LIN {X -165.856,Y 332.396,Z -10.000,A 0.015,B 0.000,C 180.000} C_DIS
LIN {X -166.589,Y 332.890,Z -10.000,A 0.015,B 0.000,C -180.000} C_DIS
LIN {X -177.836,Y 338.486,Z -10.000,A 0.015,B -0.000,C -180.000} C_DIS
LIN {X -178.207,Y 338.644,Z -10.000,A 0.015,B -0.000,C 180.000} C_DIS
LIN {X -178.933,Y 338.902,Z -10.000,A 0.015,B 0.000,C -180.000} C_DIS
LIN {X -179.548,Y 339.058,Z -10.000,A 0.015,B 0.000,C -180.000} C_DIS
LIN {X -180.489,Y 339.204,Z -10.000,A 0.015,B 0.000,C 180.000} C_DIS
LIN {X 4.865,Y 339.209,Z -10.000,A 0.015,B 0.000,C 180.000} C_DIS
LIN {X 5.937,Y 339.152,Z -10.000,A 0.015,B 0.000,C 180.000} C_DIS
LIN {X 6.802,Y 338.955,Z -10.000,A 0.015,B 0.000,C 180.000} C_DIS
LIN {X 7.069,Y 338.840,Z -10.000,A 0.015,B 0.000,C 180.000} C_DIS
LIN {X 7.566,Y 338.456,Z -9.830,A 0.015,B 0.000,C -180.000} C_DIS
LIN {X 7.779,Y 338.046,Z -9.365,A 0.015,B 0.000,C -180.000} C_DIS
LIN {X 7.818,Y 337.880,Z -8.730,A 0.015,B -0.000,C 180.000} C_DIS
$VEL.CP = 1.00000
LIN {X 7.818,Y 337.880,Z 11.000,A 0.015,B -0.000,C 180.000} C_DIS
$VEL.CP = 1.00000
LIN {X 10.265,Y 334.347,Z 11.000,A 0.015,B -0.000,C -180.000} C_DIS
$VEL.CP = 0.10000
LIN {X 10.265,Y 334.347,Z -10.000,A 0.015,B 0.000,C 180.000} C_DIS
LIN {X 10.273,Y 31.575,Z -10.000,A 0.015,B 0.000,C 180.000} C_DIS
LIN {X 8.895,Y 37.171,Z -10.000,A 0.015,B 0.000,C 180.000} C_DIS
LIN {X 8.758,Y 37.599,Z -10.000,A 0.015,B 0.000,C 180.000} C_DIS
LIN {X 8.488,Y 38.288,Z -10.000,A 0.015,B 0.000,C 180.000} C_DIS
LIN {X 8.227,Y 38.812,Z -10.000,A 0.015,B -0.000,C -180.000} C_DIS
LIN {X 2.036,Y 48.951,Z -10.000,A 0.015,B 0.000,C 180.000} C_DIS
LIN {X 1.888,Y 49.173,Z -10.000,A 0.015,B -0.000,C 180.000} C_DIS
LIN {X 1.052,Y 50.326,Z -10.000,A 0.015,B 0.000,C -180.000} C_DIS
LIN {X 0.431,Y 50.979,Z -10.000,A 0.015,B 0.000,C 180.000} C_DIS
LIN {X -7.440,Y 57.297,Z -10.000,A 0.015,B 0.000,C -180.000} C_DIS
LIN {X -7.815,Y 57.559,Z -10.000,A 0.015,B 0.000,C 180.000} C_DIS
LIN {X -8.485,Y 57.962,Z -10.000,A 0.015,B 0.000,C -180.000} C_DIS
LIN {X -9.252,Y 58.301,Z -10.000,A 0.015,B 0.000,C 180.000} C_DIS
LIN {X -19.103,Y 61.267,Z -10.000,A 0.015,B 0.000,C -180.000} C_DIS
LIN {X -19.948,Y 61.408,Z -10.000,A 0.015,B -0.000,C -180.000} C_DIS
LIN {X -21.762,Y 61.478,Z -10.000,A 0.015,B 0.000,C -180.000} C_DIS
LIN {X -22.200,Y 61.466,Z -10.000,A 0.015,B -0.000,C -180.000} C_DIS
LIN {X -29.456,Y 60.802,Z -10.000,A 0.015,B -0.000,C -180.000} C_DIS
LIN {X -29.688,Y 60.773,Z -10.000,A 0.015,B 0.000,C 180.000} C_DIS
LIN {X -31.502,Y 60.480,Z -10.000,A 0.015,B 0.000,C 180.000} C_DIS
LIN {X -32.206,Y 60.286,Z -10.000,A 0.015,B 0.000,C 180.000} C_DIS
LIN {X -34.020,Y 59.568,Z -10.000,A 0.015,B 0.000,C 180.000} C_DIS
LIN {X -34.313,Y 59.436,Z -10.000,A 0.015,B 0.000,C 180.000} C_DIS
LIN {X -41.056,Y 55.994,Z -10.000,A 0.015,B 0.000,C -180.000} C_DIS
LIN {X -41.306,Y 55.853,Z -10.000,A 0.015,B 0.000,C -180.000} C_DIS
LIN {X -42.245,Y 55.268,Z -10.000,A 0.015,B 0.000,C 180.000} C_DIS
LIN {X -42.603,Y 55.011,Z -10.000,A 0.015,B -0.000,C 180.000} C_DIS
LIN {X -43.629,Y 54.169,Z -10.000,A 0.015,B 0.000,C 180.000} C_DIS
LIN {X -44.021,Y 53.790,Z -10.000,A 0.015,B -0.000,C 180.000} C_DIS
LIN {X -46.923,Y 50.493,Z -10.000,A 0.015,B 0.000,C -180.000} C_DIS
LIN {X -46.984,Y 50.423,Z -10.000,A 0.015,B 0.000,C -180.000} C_DIS
LIN {X -50.315,Y 46.422,Z -10.000,A 0.015,B 0.000,C -180.000} C_DIS
LIN {X -50.645,Y 45.950,Z -10.000,A 0.015,B 0.000,C -180.000} C_DIS
LIN {X -68.582,Y 14.913,Z -10.000,A 0.015,B 0.000,C -180.000} C_DIS
LIN {X -68.710,Y 14.669,Z -10.000,A 0.015,B -0.000,C 180.000} C_DIS
LIN {X -69.398,Y 13.218,Z -10.000,A 0.015,B 0.000,C 180.000} C_DIS
LIN {X -69.532,Y 12.892,Z -10.000,A 0.015,B 0.000,C 180.000} C_DIS
LIN {X -72.086,Y 5.638,Z -10.000,A 0.015,B 0.000,C 180.000} C_DIS
LIN {X -72.157,Y 5.411,Z -10.000,A 0.015,B 0.000,C -180.000} C_DIS
LIN {X -72.555,Y 3.960,Z -10.000,A 0.015,B 0.000,C -180.000} C_DIS
LIN {X -72.656,Y 3.432,Z -10.000,A 0.015,B 0.000,C 180.000} C_DIS
LIN {X -72.815,Y 1.981,Z -10.000,A 0.015,B 0.000,C -180.000} C_DIS
LIN {X -72.832,Y 1.451,Z -10.000,A 0.015,B 0.000,C -180.000} C_DIS
LIN {X -72.484,Y -5.804,Z -10.000,A 0.015,B -0.000,C 180.000} C_DIS
LIN {X -72.471,Y -5.978,Z -10.000,A 0.015,B 0.000,C 180.000} C_DIS
LIN {X -72.255,Y -8.154,Z -10.000,A 0.015,B 0.000,C -180.000} C_DIS
LIN {X -72.121,Y -8.815,Z -10.000,A 0.015,B 0.000,C -180.000} C_DIS
LIN {X -71.696,Y -10.196,Z -10.000,A 0.015,B 0.000,C 180.000} C_DIS
LIN {X -71.562,Y -10.556,Z -10.000,A 0.015,B 0.000,C -180.000} C_DIS
LIN {X -70.702,Y -12.522,Z -10.000,A 0.015,B 0.000,C -180.000} C_DIS
LIN {X -70.675,Y -12.581,Z -10.000,A 0.015,B -0.000,C 180.000} C_DIS
LIN {X -68.540,Y -17.215,Z -10.000,A 0.015,B 0.000,C 180.000} C_DIS
LIN {X -68.479,Y -17.341,Z -10.000,A 0.015,B 0.000,C -180.000} C_DIS
LIN {X -67.736,Y -18.792,Z -10.000,A 0.015,B 0.000,C 180.000} C_DIS
LIN {X -67.504,Y -19.179,Z -10.000,A 0.015,B 0.000,C -180.000} C_DIS
LIN {X -66.730,Y -20.294,Z -10.000,A 0.015,B 0.000,C -180.000} C_DIS
LIN {X -66.274,Y -20.824,Z -10.000,A 0.015,B -0.000,C 180.000} C_DIS
LIN {X -59.767,Y -26.968,Z -10.000,A 0.015,B 0.000,C 180.000} C_DIS
LIN {X -59.610,Y -27.107,Z -10.000,A 0.015,B 0.000,C 180.000} C_DIS
LIN {X -58.521,Y -28.014,Z -10.000,A 0.015,B 0.000,C 180.000} C_DIS
CIRC {X -58.086,Y -28.321,Z -10.000,A 0.015,B 0.000,C 180.000},{X -57.609,Y -28.557,Z -10.000,A 0.015,B 0.000,C 180.000} C_DIS
LIN {X -50.808,Y -31.266,Z -10.000,A 0.015,B 0.000,C 180.000} C_DIS
LIN {X -342.732,Y -31.266,Z -10.000,A 0.015,B 0.000,C -180.000} C_DIS
LIN {X -336.289,Y -28.753,Z -10.000,A 0.015,B 0.000,C 180.000} C_DIS
LIN {X -335.780,Y -28.504,Z -10.000,A 0.015,B -0.000,C 180.000} C_DIS
LIN {X -335.055,Y -28.070,Z -10.000,A 0.015,B 0.000,C -180.000} C_DIS
LIN {X -334.490,Y -27.645,Z -10.000,A 0.015,B -0.000,C -180.000} C_DIS
LIN {X -332.313,Y -25.623,Z -10.000,A 0.015,B 0.000,C 180.000} C_DIS
LIN {X -332.274,Y -25.586,Z -10.000,A 0.015,B -0.000,C -180.000} C_DIS
LIN {X -326.917,Y -20.448,Z -10.000,A 0.015,B 0.000,C 180.000} C_DIS
LIN {X -326.374,Y -19.773,Z -10.000,A 0.015,B -0.000,C 180.000} C_DIS
LIN {X -325.688,Y -18.654,Z -10.000,A 0.015,B -0.000,C 180.000} C_DIS
LIN {X -325.506,Y -18.313,Z -10.000,A 0.015,B 0.000,C 180.000} C_DIS
LIN {X -322.238,Y -11.280,Z -10.000,A 0.015,B 0.000,C 180.000} C_DIS
LIN {X -322.125,Y -11.006,Z -10.000,A 0.015,B 0.000,C -180.000} C_DIS
LIN {X -321.519,Y -9.333,Z -10.000,A 0.015,B 0.000,C -180.000} C_DIS
LIN {X -321.339,Y -8.569,Z -10.000,A 0.015,B -0.000,C -180.000} C_DIS
LIN {X -321.046,Y -6.030,Z -10.000,A 0.015,B 0.000,C -180.000} C_DIS
LIN {X -321.028,Y -5.804,Z -10.000,A 0.015,B -0.000,C -180.000} C_DIS
LIN {X -320.680,Y 1.451,Z -10.000,A 0.015,B 0.000,C 180.000} C_DIS
LIN {X -320.686,Y 1.861,Z -10.000,A 0.015,B 0.000,C -180.000} C_DIS
LIN {X -320.739,Y 2.586,Z -10.000,A 0.015,B -0.000,C -180.000} C_DIS
LIN {X -320.784,Y 2.941,Z -10.000,A 0.015,B -0.000,C -180.000} C_DIS
LIN {X -321.047,Y 4.392,Z -10.000,A 0.015,B -0.000,C 180.000} C_DIS
LIN {X -321.174,Y 4.882,Z -10.000,A 0.015,B 0.000,C -180.000} C_DIS
LIN {X -321.917,Y 7.058,Z -10.000,A 0.015,B 0.000,C 180.000} C_DIS
LIN {X -321.936,Y 7.114,Z -10.000,A 0.015,B -0.000,C 180.000} C_DIS
LIN {X -324.293,Y 13.643,Z -10.000,A 0.015,B 0.000,C 180.000} C_DIS
LIN {X -324.544,Y 14.184,Z -10.000,A 0.015,B 0.000,C -180.000} C_DIS
LIN {X -342.520,Y 45.380,Z -10.000,A 0.015,B -0.000,C -180.000} C_DIS
LIN {X -342.658,Y 45.599,Z -10.000,A 0.015,B 0.000,C 180.000} C_DIS
LIN {X -343.432,Y 46.732,Z -10.000,A 0.015,B -0.000,C 180.000} C_DIS
LIN {X -343.654,Y 47.022,Z -10.000,A 0.015,B 0.000,C -180.000} C_DIS
LIN {X -348.970,Y 53.238,Z -10.000,A 0.015,B 0.000,C 180.000} C_DIS
LIN {X -349.184,Y 53.466,Z -10.000,A 0.015,B 0.000,C 180.000} C_DIS
LIN {X -350.186,Y 54.439,Z -10.000,A 0.015,B 0.000,C 180.000} C_DIS
LIN {X -350.569,Y 54.760,Z -10.000,A 0.015,B 0.000,C -180.000} C_DIS
LIN {X -351.551,Y 55.465,Z -10.000,A 0.015,B 0.000,C 180.000} C_DIS
LIN {X -351.978,Y 55.726,Z -10.000,A 0.015,B 0.000,C -180.000} C_DIS
LIN {X -359.191,Y 59.432,Z -10.000,A 0.015,B 0.000,C -180.000} C_DIS
LIN {X -359.413,Y 59.536,Z -10.000,A 0.015,B 0.000,C -180.000} C_DIS
LIN {X -360.864,Y 60.153,Z -10.000,A 0.015,B -0.000,C 180.000} C_DIS
LIN {X -361.495,Y 60.351,Z -10.000,A 0.015,B 0.000,C -180.000} C_DIS
LIN {X -362.947,Y 60.654,Z -10.000,A 0.015,B 0.000,C 180.000} C_DIS
LIN {X -363.320,Y 60.711,Z -10.000,A 0.015,B 0.000,C 180.000} C_DIS
LIN {X -371.302,Y 61.465,Z -10.000,A 0.015,B 0.000,C -180.000} C_DIS
LIN {X -371.750,Y 61.478,Z -10.000,A 0.015,B 0.000,C -180.000} C_DIS
LIN {X -373.564,Y 61.408,Z -10.000,A 0.015,B -0.000,C 180.000} C_DIS
LIN {X -374.398,Y 61.270,Z -10.000,A 0.015,B -0.000,C -180.000} C_DIS
LIN {X -383.578,Y 58.541,Z -10.000,A 0.015,B 0.000,C -180.000} C_DIS
LIN {X -383.897,Y 58.428,Z -10.000,A 0.015,B 0.000,C 180.000} C_DIS
LIN {X -384.902,Y 58.016,Z -10.000,A 0.015,B 0.000,C 180.000} C_DIS
LIN {X -385.717,Y 57.540,Z -10.000,A 0.015,B -0.000,C 180.000} C_DIS
LIN {X -393.232,Y 51.598,Z -10.000,A 0.015,B 0.000,C -180.000} C_DIS
LIN {X -393.470,Y 51.391,Z -10.000,A 0.015,B -0.000,C 180.000} C_DIS
LIN {X -394.404,Y 50.499,Z -10.000,A 0.015,B 0.000,C -180.000} C_DIS
LIN {X -394.942,Y 49.837,Z -10.000,A 0.015,B -0.000,C 180.000} C_DIS
LIN {X -401.253,Y 39.671,Z -10.000,A 0.015,B 0.000,C 180.000} C_DIS
LIN {X -401.377,Y 39.454,Z -10.000,A 0.015,B 0.000,C 180.000} C_DIS
LIN {X -401.994,Y 38.272,Z -10.000,A 0.015,B 0.000,C -180.000} C_DIS
LIN {X -402.274,Y 37.542,Z -10.000,A 0.015,B -0.000,C 180.000} C_DIS
LIN {X -403.779,Y 31.645,Z -10.000,A 0.015,B 0.000,C 180.000} C_DIS
LIN {X -403.787,Y 333.800,Z -10.000,A 0.015,B 0.000,C 180.000} C_DIS
LIN {X -403.730,Y 334.871,Z -10.000,A 0.015,B -0.000,C -180.000} C_DIS
LIN {X -403.533,Y 335.736,Z -10.000,A 0.015,B 0.000,C -180.000} C_DIS
LIN {X -403.418,Y 336.003,Z -10.000,A 0.015,B -0.000,C -180.000} C_DIS
LIN {X -403.034,Y 336.500,Z -9.830,A 0.015,B 0.000,C -180.000} C_DIS
LIN {X -402.624,Y 336.714,Z -9.365,A 0.015,B -0.000,C -180.000} C_DIS
LIN {X -402.458,Y 336.753,Z -8.730,A 0.015,B 0.000,C -180.000} C_DIS
$VEL.CP = 1.00000
LIN {X -402.458,Y 336.753,Z 11.000,A 0.015,B 0.000,C 180.000} C_DIS
$VEL.CP = 1.00000
LIN {X -182.199,Y 109.361,Z 11.000,A 0.015,B 0.000,C 180.000} C_DIS
$VEL.CP = 1.00000
LIN {X -182.199,Y 109.361,Z 1.769,A 0.015,B -0.000,C 180.000} C_DIS
$VEL.CP = 0.10000
LIN {X -182.037,Y 109.343,Z 1.147,A 0.015,B 0.000,C 180.000} C_DIS
LIN {X -181.592,Y 109.314,Z 0.684,A 0.015,B -0.000,C -180.000} C_DIS
LIN {X -180.976,Y 109.330,Z 0.500,A 0.015,B 0.000,C -180.000} C_DIS
LIN {X -175.739,Y 113.354,Z 0.256,A 0.015,B 0.000,C -180.000} C_DIS
LIN {X -177.328,Y 119.764,Z 0.012,A 0.015,B 0.000,C 180.000} C_DIS
LIN {X -183.837,Y 120.878,Z -0.232,A 0.015,B 0.000,C -180.000} C_DIS
LIN {X -187.466,Y 115.360,Z -0.476,A 0.015,B -0.000,C -180.000} C_DIS
LIN {X -183.865,Y 109.824,Z -0.720,A 0.015,B 0.000,C -180.000} C_DIS
LIN {X -177.349,Y 110.905,Z -0.964,A 0.015,B 0.000,C -180.000} C_DIS
LIN {X -175.729,Y 117.308,Z -1.208,A 0.015,B 0.000,C -180.000} C_DIS
LIN {X -180.946,Y 121.358,Z -1.452,A 0.015,B 0.000,C -180.000} C_DIS
LIN {X -186.747,Y 118.201,Z -1.696,A 0.015,B 0.000,C -180.000} C_DIS
LIN {X -186.180,Y 111.621,Z -1.940,A 0.015,B 0.000,C -180.000} C_DIS
LIN {X -179.924,Y 109.504,Z -2.185,A 0.015,B 0.000,C 180.000} C_DIS
LIN {X -175.478,Y 114.388,Z -2.429,A 0.015,B -0.000,C -180.000} C_DIS
LIN {X -178.170,Y 120.418,Z -2.673,A 0.015,B 0.000,C 180.000} C_DIS
LIN {X -184.774,Y 120.368,Z -2.917,A 0.015,B 0.000,C 180.000} C_DIS
LIN {X -187.374,Y 114.297,Z -3.161,A 0.015,B -0.000,C 180.000} C_DIS
LIN {X -182.854,Y 109.482,Z -3.405,A 0.015,B 0.000,C -180.000} C_DIS
LIN {X -176.631,Y 111.694,Z -3.649,A 0.015,B 0.000,C -180.000} C_DIS
LIN {X -176.164,Y 118.282,Z -3.893,A 0.015,B 0.000,C 180.000} C_DIS
LIN {X -182.013,Y 121.350,Z -4.137,A 0.015,B 0.000,C 180.000} C_DIS
LIN {X -187.167,Y 117.220,Z -4.381,A 0.015,B 0.000,C -180.000} C_DIS
LIN {X -185.449,Y 110.843,Z -4.625,A 0.015,B 0.000,C 180.000} C_DIS
LIN {X -178.919,Y 109.862,Z -4.869,A 0.015,B -0.000,C -180.000} C_DIS
LIN {X -175.402,Y 115.452,Z -5.113,A 0.015,B 0.000,C 180.000} C_DIS
LIN {X -179.115,Y 120.914,Z -5.357,A 0.015,B 0.000,C -180.000} C_DIS
LIN {X -185.607,Y 119.701,Z -5.601,A 0.015,B 0.000,C 180.000} C_DIS
LIN {X -187.097,Y 113.267,Z -5.845,A 0.015,B 0.000,C -180.000} C_DIS
LIN {X -181.799,Y 109.324,Z -6.089,A 0.015,B 0.000,C -180.000} C_DIS
LIN {X -176.063,Y 112.597,Z -6.333,A 0.015,B 0.000,C -180.000} C_DIS
LIN {X -176.764,Y 119.164,Z -6.577,A 0.015,B 0.000,C -180.000} C_DIS
LIN {X -183.061,Y 121.154,Z -6.821,A 0.015,B 0.000,C 180.000} C_DIS
LIN {X -187.408,Y 116.181,Z -7.065,A 0.015,B 0.000,C 180.000} C_DIS
LIN {X -184.594,Y 110.206,Z -7.310,A 0.015,B 0.000,C -180.000} C_DIS
LIN {X -177.992,Y 110.390,Z -7.554,A 0.015,B 0.000,C -180.000} C_DIS
LIN {X -175.515,Y 116.513,Z -7.798,A 0.015,B -0.000,C 180.000} C_DIS
LIN {X -180.132,Y 121.235,Z -8.042,A 0.015,B 0.000,C -180.000} C_DIS
LIN {X -186.309,Y 118.898,Z -8.286,A 0.015,B 0.000,C 180.000} C_DIS
LIN {X -186.643,Y 112.302,Z -8.530,A 0.015,B -0.000,C 180.000} C_DIS
LIN {X -180.733,Y 109.353,Z -8.774,A 0.015,B 0.000,C 180.000} C_DIS
LIN {X -175.663,Y 113.586,Z -9.018,A 0.015,B -0.000,C -180.000} C_DIS
LIN {X -177.510,Y 119.927,Z -9.262,A 0.015,B 0.000,C 180.000} C_DIS
LIN {X -184.059,Y 120.776,Z -9.506,A 0.015,B 0.000,C -180.000} C_DIS
LIN {X -187.462,Y 115.116,Z -9.750,A 0.015,B 0.000,C -180.000} C_DIS
LIN {X -183.639,Y 109.730,Z -9.994,A 0.015,B 0.000,C 180.000} C_DIS
LIN {X -177.173,Y 111.074,Z -10.238,A 0.015,B 0.000,C 180.000} C_DIS
LIN {X -175.813,Y 117.537,Z -10.482,A 0.015,B 0.000,C 180.000} C_DIS
LIN {X -181.190,Y 121.373,Z -10.726,A 0.015,B 0.000,C -180.000} C_DIS
LIN {X -186.858,Y 117.984,Z -10.970,A 0.015,B 0.000,C 180.000} C_DIS
LIN {X -186.025,Y 111.432,Z -11.214,A 0.015,B -0.000,C -180.000} C_DIS
LIN {X -179.689,Y 109.570,Z -11.458,A 0.015,B 0.000,C -180.000} C_DIS
LIN {X -175.444,Y 114.630,Z -11.702,A 0.015,B 0.000,C 180.000} C_DIS
LIN {X -178.378,Y 120.546,Z -11.946,A 0.015,B 0.000,C -180.000} C_DIS
LIN {X -184.975,Y 120.229,Z -12.190,A 0.015,B 0.000,C 180.000} C_DIS
LIN {X -187.327,Y 114.058,Z -12.435,A 0.015,B -0.000,C -180.000} C_DIS
LIN {X -182.616,Y 109.429,Z -12.679,A 0.015,B -0.000,C -180.000} C_DIS
LIN {X -176.488,Y 111.891,Z -12.923,A 0.015,B -0.000,C -180.000} C_DIS
LIN {X -176.287,Y 118.492,Z -13.167,A 0.015,B 0.000,C 180.000} C_DIS
LIN {X -182.255,Y 121.321,Z -13.411,A 0.015,B 0.000,C -180.000} C_DIS
LIN {X -187.238,Y 116.987,Z -13.655,A 0.015,B 0.000,C 180.000} C_DIS
LIN {X -185.264,Y 110.685,Z -13.899,A 0.015,B -0.000,C -180.000} C_DIS
LIN {X -178.699,Y 109.968,Z -14.143,A 0.015,B 0.000,C -180.000} C_DIS
LIN {X -175.411,Y 115.696,Z -14.387,A 0.015,B -0.000,C 180.000} C_DIS
LIN {X -179.342,Y 121.003,Z -14.631,A 0.015,B -0.000,C 180.000} C_DIS
LIN {X -185.780,Y 119.529,Z -14.875,A 0.015,B 0.000,C -180.000} C_DIS
LIN {X -187.008,Y 113.040,Z -15.119,A 0.015,B -0.000,C 180.000} C_DIS
LIN {X -181.556,Y 109.314,Z -15.363,A 0.015,B 0.000,C 180.000} C_DIS
LIN {X -175.957,Y 112.816,Z -15.607,A 0.015,B 0.000,C -180.000} C_DIS
LIN {X -176.922,Y 119.350,Z -15.851,A 0.015,B -0.000,C -180.000} C_DIS
LIN {X -183.295,Y 121.083,Z -16.095,A 0.015,B 0.000,C 180.000} C_DIS
LIN {X -187.437,Y 115.939,Z -16.339,A 0.015,B 0.000,C 180.000} C_DIS
LIN {X -184.384,Y 110.083,Z -16.583,A 0.015,B -0.000,C 180.000} C_DIS
LIN {X -177.795,Y 110.534,Z -16.827,A 0.015,B 0.000,C 180.000} C_DIS
LIN {X -175.567,Y 116.751,Z -17.071,A 0.015,B 0.000,C -180.000} C_DIS
LIN {X -180.371,Y 121.283,Z -17.315,A 0.015,B -0.000,C 180.000} C_DIS
LIN {X -186.448,Y 118.698,Z -17.560,A 0.015,B 0.000,C -180.000} C_DIS
LIN {X -186.515,Y 112.094,Z -17.804,A 0.015,B 0.000,C -180.000} C_DIS
LIN {X -180.491,Y 109.386,Z -18.048,A 0.015,B -0.000,C 180.000} C_DIS
LIN {X -175.597,Y 113.821,Z -18.292,A 0.015,B 0.000,C -180.000} C_DIS
LIN {X -177.698,Y 120.082,Z -18.536,A 0.015,B 0.000,C 180.000} C_DIS
LIN {X -184.277,Y 120.666,Z -18.780,A 0.015,B -0.000,C 180.000} C_DIS
LIN {X -187.448,Y 114.872,Z -19.024,A 0.015,B 0.000,C 180.000} C_DIS
LIN {X -183.411,Y 109.646,Z -19.268,A 0.015,B -0.000,C -180.000} C_DIS
LIN {X -177.004,Y 111.250,Z -19.512,A 0.015,B -0.000,C 180.000} C_DIS
LIN {X -175.907,Y 117.762,Z -19.756,A 0.015,B 0.000,C 180.000} C_DIS
LIN {X -181.434,Y 121.377,Z -20.000,A 0.015,B 0.000,C -180.000} C_DIS
LIN {X -213.976,Y 121.377,Z -20.000,A 0.015,B 0.000,C 180.000} C_DIS
CIRC {X -215.901,Y 120.266,Z -20.000,A 0.015,B 0.000,C 180.000},{X -215.902,Y 118.044,Z -20.000,A 0.015,B 0.000,C -180.000} C_DIS
LIN {X -214.807,Y 116.142,Z -20.000,A 0.015,B 0.000,C 180.000} C_DIS
CIRC {X -213.767,Y 115.102,Z -20.000,A 0.015,B 0.000,C 180.000},{X -212.347,Y 114.721,Z -20.000,A 0.015,B 0.000,C -180.000} C_DIS
LIN {X -181.151,Y 114.721,Z -20.000,A 0.015,B 0.000,C 180.000} C_DIS
CIRC {X -179.732,Y 115.101,Z -20.000,A 0.015,B 0.000,C 180.000},{X -178.693,Y 116.139,Z -20.000,A 0.015,B 0.000,C 180.000} C_DIS
LIN {X -177.595,Y 118.039,Z -20.000,A 0.015,B -0.000,C 180.000} C_DIS
CIRC {X -177.595,Y 120.265,Z -20.000,A 0.015,B 0.000,C 180.000},{X -179.522,Y 121.377,Z -20.000,A 0.015,B -0.000,C 180.000} C_DIS
LIN {X -181.434,Y 121.377,Z -20.000,A 0.015,B 0.000,C -180.000} C_DIS
CIRC {X -184.808,Y 122.399,Z -20.000,A 0.015,B 0.000,C 180.000},{X -187.049,Y 125.121,Z -20.000,A 0.015,B 0.000,C 180.000} C_DIS
CIRC {X -189.290,Y 127.843,Z -20.000,A 0.015,B 0.000,C 180.000},{X -192.665,Y 128.864,Z -20.000,A 0.015,B 0.000,C 180.000} C_DIS
LIN {X -214.895,Y 128.864,Z -20.000,A 0.015,B -0.000,C 180.000} C_DIS
CIRC {X -218.571,Y 128.969,Z -20.000,A 0.015,B 0.000,C -180.000},{X -222.234,Y 129.283,Z -20.000,A 0.015,B 0.000,C -180.000} C_DIS
CIRC {X -225.886,Y 129.692,Z -20.000,A 0.015,B 0.000,C 180.000},{X -229.541,Y 130.082,Z -20.000,A 0.015,B 0.000,C 180.000} C_DIS
CIRC {X -231.339,Y 129.164,Z -20.000,A 0.015,B 0.000,C -180.000},{X -231.232,Y 127.147,Z -20.000,A 0.015,B 0.000,C -180.000} C_DIS
CIRC {X -228.499,Y 123.234,Z -20.000,A 0.015,B 0.000,C 180.000},{X -225.916,Y 119.220,Z -20.000,A 0.015,B 0.000,C 180.000} C_DIS
CIRC {X -223.440,Y 115.140,Z -20.000,A 0.015,B 0.000,C 180.000},{X -221.026,Y 111.023,Z -20.000,A 0.015,B -0.000,C 180.000} C_DIS
CIRC {X -217.921,Y 107.915,Z -20.000,A 0.015,B 0.000,C 180.000},{X -213.677,Y 106.777,Z -20.000,A 0.015,B -0.000,C 180.000} C_DIS
LIN {X -179.835,Y 106.777,Z -20.000,A 0.015,B 0.000,C -180.000} C_DIS
CIRC {X -175.585,Y 107.915,Z -20.000,A 0.015,B -0.000,C -180.000},{X -172.474,Y 111.024,Z -20.000,A 0.015,B 0.000,C 180.000} C_DIS
CIRC {X -170.062,Y 115.134,Z -20.000,A 0.015,B 0.000,C -180.000},{X -167.597,Y 119.212,Z -20.000,A 0.015,B 0.000,C -180.000} C_DIS
CIRC {X -165.028,Y 123.227,Z -20.000,A 0.015,B -0.000,C 180.000},{X -162.308,Y 127.141,Z -20.000,A 0.015,B 0.000,C 180.000} C_DIS
CIRC {X -162.205,Y 129.160,Z -20.000,A 0.015,B 0.000,C 180.000},{X -164.006,Y 130.079,Z -20.000,A 0.015,B -0.000,C 180.000} C_DIS
CIRC {X -167.652,Y 129.690,Z -20.000,A 0.015,B -0.000,C 180.000},{X -171.295,Y 129.283,Z -20.000,A 0.015,B 0.000,C 180.000} C_DIS
CIRC {X -174.950,Y 128.969,Z -20.000,A 0.015,B -0.000,C 180.000},{X -178.617,Y 128.865,Z -20.000,A 0.015,B 0.000,C -180.000} C_DIS
LIN {X -192.665,Y 128.864,Z -20.000,A 0.015,B 0.000,C -180.000} C_DIS
CIRC {X -195.950,Y 129.859,Z -20.000,A 0.015,B 0.000,C -180.000},{X -198.132,Y 132.509,Z -20.000,A 0.015,B 0.000,C 180.000} C_DIS
CIRC {X -200.314,Y 135.159,Z -20.000,A 0.015,B 0.000,C 180.000},{X -203.599,Y 136.154,Z -20.000,A 0.015,B 0.000,C 180.000} C_DIS
LIN {X -214.895,Y 136.154,Z -20.000,A 0.015,B 0.000,C -180.000} C_DIS
CIRC {X -223.130,Y 136.478,Z -20.000,A 0.015,B 0.000,C 180.000},{X -231.314,Y 137.447,Z -20.000,A 0.015,B -0.000,C -180.000} C_DIS
CIRC {X -239.436,Y 138.810,Z -20.000,A 0.015,B 0.000,C -180.000},{X -247.532,Y 140.318,Z -20.000,A 0.015,B -0.000,C 180.000} C_DIS
CIRC {X -249.264,Y 139.531,Z -20.000,A 0.015,B 0.000,C 180.000},{X -249.086,Y 137.637,Z -20.000,A 0.015,B -0.000,C 180.000} C_DIS
CIRC {X -243.729,Y 131.288,Z -20.000,A 0.015,B -0.000,C 180.000},{X -238.530,Y 124.808,Z -20.000,A 0.015,B 0.000,C 180.000} C_DIS
CIRC {X -233.643,Y 118.085,Z -20.000,A 0.015,B 0.000,C -180.000},{X -229.242,Y 111.034,Z -20.000,A 0.015,B 0.000,C 180.000} C_DIS
CIRC {X -228.225,Y 109.203,Z -20.000,A 0.015,B 0.000,C -180.000},{X -227.265,Y 107.341,Z -20.000,A 0.015,B 0.000,C -180.000} C_DIS
CIRC {X -226.305,Y 105.479,Z -20.000,A 0.015,B 0.000,C 180.000},{X -225.288,Y 103.648,Z -20.000,A 0.015,B 0.000,C 180.000} C_DIS
CIRC {X -222.183,Y 100.539,Z -20.000,A 0.015,B 0.000,C -180.000},{X -217.939,Y 99.401,Z -20.000,A 0.015,B -0.000,C -180.000} C_DIS
LIN {X -175.579,Y 99.401,Z -20.000,A 0.015,B 0.000,C 180.000} C_DIS
CIRC {X -171.329,Y 100.540,Z -20.000,A 0.015,B -0.000,C 180.000},{X -168.218,Y 103.649,Z -20.000,A 0.015,B 0.000,C -180.000} C_DIS
CIRC {X -167.137,Y 105.588,Z -20.000,A 0.015,B 0.000,C -180.000},{X -166.118,Y 107.559,Z -20.000,A 0.015,B 0.000,C -180.000} C_DIS
CIRC {X -165.099,Y 109.531,Z -20.000,A 0.015,B 0.000,C 180.000},{X -164.019,Y 111.469,Z -20.000,A 0.015,B -0.000,C -180.000} C_DIS
CIRC {X -159.670,Y 118.415,Z -20.000,A 0.015,B 0.000,C 180.000},{X -154.841,Y 125.037,Z -20.000,A 0.015,B 0.000,C 180.000} C_DIS
CIRC {X -149.698,Y 131.412,Z -20.000,A 0.015,B 0.000,C 180.000},{X -144.387,Y 137.648,Z -20.000,A 0.015,B 0.000,C 180.000} C_DIS
CIRC {X -144.201,Y 139.539,Z -20.000,A 0.015,B 0.000,C 180.000},{X -145.931,Y 140.327,Z -20.000,A 0.015,B 0.000,C -180.000} C_DIS
CIRC {X -154.039,Y 138.817,Z -20.000,A 0.015,B 0.000,C 180.000},{X -162.173,Y 137.451,Z -20.000,A 0.015,B 0.000,C 180.000} C_DIS
CIRC {X -170.369,Y 136.479,Z -20.000,A 0.015,B -0.000,C -180.000},{X -178.617,Y 136.154,Z -20.000,A 0.015,B -0.000,C -180.000} C_DIS
LIN {X -203.599,Y 136.154,Z -20.000,A 0.015,B 0.000,C 180.000} C_DIS
CIRC {X -206.696,Y 137.092,Z -20.000,A 0.015,B 0.000,C 180.000},{X -208.752,Y 139.589,Z -20.000,A 0.015,B -0.000,C 180.000} C_DIS
CIRC {X -210.808,Y 142.086,Z -20.000,A 0.015,B 0.000,C -180.000},{X -213.904,Y 143.024,Z -20.000,A 0.015,B -0.000,C 180.000} C_DIS
LIN {X -214.895,Y 143.024,Z -20.000,A 0.015,B -0.000,C -180.000} C_DIS
CIRC {X -230.200,Y 143.852,Z -20.000,A 0.015,B -0.000,C 180.000},{X -245.325,Y 146.329,Z -20.000,A 0.015,B 0.000,C 180.000} C_DIS
CIRC {X -260.127,Y 150.280,Z -20.000,A 0.015,B 0.000,C -180.000},{X -274.518,Y 155.531,Z -20.000,A 0.015,B 0.000,C -180.000} C_DIS
CIRC {X -276.076,Y 155.002,Z -20.000,A 0.015,B 0.000,C 180.000},{X -275.748,Y 153.390,Z -20.000,A 0.015,B 0.000,C 180.000} C_DIS
CIRC {X -266.780,Y 146.054,Z -20.000,A 0.015,B 0.000,C 180.000},{X -258.385,Y 138.068,Z -20.000,A 0.015,B -0.000,C -180.000} C_DIS
CIRC {X -250.572,Y 129.516,Z -20.000,A 0.015,B 0.000,C -180.000},{X -243.334,Y 120.471,Z -20.000,A 0.015,B -0.000,C 180.000} C_DIS
CIRC {X -241.113,Y 117.375,Z -20.000,A 0.015,B 0.000,C 180.000},{X -239.019,Y 114.192,Z -20.000,A 0.015,B 0.000,C 180.000} C_DIS
CIRC {X -237.021,Y 110.948,Z -20.000,A 0.015,B 0.000,C 180.000},{X -235.087,Y 107.666,Z -20.000,A 0.015,B 0.000,C -180.000} C_DIS
CIRC {X -233.587,Y 104.967,Z -20.000,A 0.015,B 0.000,C -180.000},{X -232.172,Y 102.222,Z -20.000,A 0.015,B 0.000,C -180.000} C_DIS
CIRC {X -230.758,Y 99.478,Z -20.000,A 0.015,B 0.000,C 180.000},{X -229.258,Y 96.779,Z -20.000,A 0.015,B 0.000,C -180.000} C_DIS
CIRC {X -226.153,Y 93.670,Z -20.000,A 0.015,B 0.000,C 180.000},{X -221.909,Y 92.532,Z -20.000,A 0.015,B 0.000,C 180.000} C_DIS
LIN {X -171.614,Y 92.532,Z -20.000,A 0.015,B -0.000,C 180.000} C_DIS
CIRC {X -167.365,Y 93.670,Z -20.000,A 0.015,B -0.000,C 180.000},{X -164.253,Y 96.779,Z -20.000,A 0.015,B 0.000,C 180.000} C_DIS
CIRC {X -162.690,Y 99.584,Z -20.000,A 0.015,B -0.000,C -180.000},{X -161.216,Y 102.437,Z -20.000,A 0.015,B 0.000,C -180.000} C_DIS
CIRC {X -159.741,Y 105.289,Z -20.000,A 0.015,B 0.000,C -180.000},{X -158.178,Y 108.094,Z -20.000,A 0.015,B 0.000,C 180.000} C_DIS
CIRC {X -149.836,Y 120.906,Z -20.000,A 0.015,B 0.000,C -180.000},{X -140.182,Y 132.761,Z -20.000,A 0.015,B 0.000,C 180.000} C_DIS
CIRC {X -129.413,Y 143.604,Z -20.000,A 0.015,B -0.000,C -180.000},{X -117.706,Y 153.428,Z -20.000,A 0.015,B 0.000,C 180.000} C_DIS
CIRC {X -117.387,Y 155.041,Z -20.000,A 0.015,B 0.000,C -180.000},{X -118.946,Y 155.561,Z -20.000,A 0.015,B 0.000,C -180.000} C_DIS
CIRC {X -129.295,Y 151.617,Z -20.000,A 0.015,B -0.000,C 180.000},{X -139.903,Y 148.434,Z -20.000,A 0.015,B -0.000,C 180.000} C_DIS
CIRC {X -150.698,Y 145.966,Z -20.000,A 0.015,B 0.000,C -180.000},{X -161.622,Y 144.160,Z -20.000,A 0.015,B 0.000,C 180.000} C_DIS
CIRC {X -170.100,Y 143.308,Z -20.000,A 0.015,B 0.000,C -180.000},{X -178.617,Y 143.024,Z -20.000,A 0.015,B -0.000,C 180.000} C_DIS
LIN {X -213.904,Y 143.024,Z -20.000,A 0.015,B -0.000,C -180.000} C_DIS
CIRC {X -216.881,Y 143.931,Z -20.000,A 0.015,B 0.000,C -180.000},{X -218.845,Y 146.346,Z -20.000,A 0.015,B 0.000,C -180.000} C_DIS
CIRC {X -220.762,Y 148.779,Z -20.000,A 0.015,B 0.000,C -180.000},{X -223.679,Y 149.821,Z -20.000,A 0.015,B 0.000,C 180.000} C_DIS
CIRC {X -236.972,Y 151.303,Z -20.000,A 0.015,B -0.000,C 180.000},{X -250.063,Y 154.051,Z -20.000,A 0.015,B 0.000,C 180.000} C_DIS
CIRC {X -266.963,Y 159.495,Z -20.000,A 0.015,B 0.000,C -180.000},{X -283.139,Y 166.817,Z -20.000,A 0.015,B 0.000,C -180.000} C_DIS
CIRC {X -285.396,Y 166.746,Z -20.000,A 0.015,B 0.000,C -180.000},{X -286.505,Y 164.779,Z -20.000,A 0.015,B 0.000,C -180.000} C_DIS
LIN {X -286.505,Y 156.621,Z -20.000,A 0.015,B 0.000,C -180.000} C_DIS
CIRC {X -285.744,Y 153.492,Z -20.000,A 0.015,B 0.000,C -180.000},{X -283.631,Y 151.063,Z -20.000,A 0.015,B 0.000,C 180.000} C_DIS
CIRC {X -271.089,Y 141.188,Z -20.000,A 0.015,B 0.000,C -180.000},{X -259.609,Y 130.095,Z -20.000,A 0.015,B 0.000,C -180.000} C_DIS
CIRC {X -249.387,Y 117.826,Z -20.000,A 0.015,B -0.000,C -180.000},{X -240.634,Y 104.469,Z -20.000,A 0.015,B -0.000,C 180.000} C_DIS
CIRC {X -238.677,Y 100.946,Z -20.000,A 0.015,B 0.000,C -180.000},{X -236.830,Y 97.364,Z -20.000,A 0.015,B -0.000,C -180.000} C_DIS
CIRC {X -234.984,Y 93.781,Z -20.000,A 0.015,B 0.000,C 180.000},{X -233.026,Y 90.258,Z -20.000,A 0.015,B 0.000,C -180.000} C_DIS
CIRC {X -229.921,Y 87.149,Z -20.000,A 0.015,B 0.000,C -180.000},{X -225.677,Y 86.011,Z -20.000,A 0.015,B 0.000,C -180.000} C_DIS
LIN {X -167.851,Y 86.011,Z -20.000,A 0.015,B 0.000,C 180.000} C_DIS
CIRC {X -163.602,Y 87.149,Z -20.000,A 0.015,B -0.000,C 180.000},{X -160.491,Y 90.259,Z -20.000,A 0.015,B 0.000,C -180.000} C_DIS
CIRC {X -158.469,Y 93.886,Z -20.000,A 0.015,B 0.000,C 180.000},{X -156.562,Y 97.575,Z -20.000,A 0.015,B -0.000,C 180.000} C_DIS
CIRC {X -154.655,Y 101.263,Z -20.000,A 0.015,B 0.000,C 180.000},{X -152.634,Y 104.890,Z -20.000,A 0.015,B 0.000,C 180.000} C_DIS
CIRC {X -143.933,Y 118.137,Z -20.000,A 0.015,B 0.000,C 180.000},{X -133.779,Y 130.306,Z -20.000,A 0.015,B 0.000,C 180.000} C_DIS
CIRC {X -122.371,Y 141.301,Z -20.000,A 0.015,B 0.000,C 180.000},{X -109.898,Y 151.071,Z -20.000,A 0.015,B 0.000,C -180.000} C_DIS
CIRC {X -107.773,Y 153.503,Z -20.000,A 0.015,B 0.000,C 180.000},{X -107.007,Y 156.641,Z -20.000,A 0.015,B 0.000,C -180.000} C_DIS
LIN {X -107.007,Y 164.771,Z -20.000,A 0.015,B 0.000,C -180.000} C_DIS
CIRC {X -108.116,Y 166.734,Z -20.000,A 0.015,B 0.000,C -180.000},{X -110.370,Y 166.798,Z -20.000,A 0.015,B -0.000,C -180.000} C_DIS
CIRC {X -122.792,Y 160.992,Z -20.000,A 0.015,B 0.000,C 180.000},{X -135.716,Y 156.411,Z -20.000,A 0.015,B 0.000,C -180.000} C_DIS
CIRC {X -148.988,Y 152.984,Z -20.000,A 0.015,B 0.000,C 180.000},{X -162.490,Y 150.622,Z -20.000,A 0.015,B 0.000,C 180.000} C_DIS
CIRC {X -170.535,Y 149.814,Z -20.000,A 0.015,B 0.000,C -180.000},{X -178.617,Y 149.544,Z -20.000,A 0.015,B 0.000,C -180.000} C_DIS
LIN {X -214.895,Y 149.544,Z -20.000,A 0.015,B 0.000,C -180.000} C_DIS
CIRC {X -219.289,Y 149.614,Z -20.000,A 0.015,B 0.000,C 180.000},{X -223.679,Y 149.821,Z -20.000,A 0.015,B -0.000,C 180.000} C_DIS
CIRC {X -227.301,Y 151.186,Z -20.000,A 0.015,B 0.000,C 180.000},{X -229.536,Y 154.346,Z -20.000,A 0.015,B -0.000,C 180.000} C_DIS
CIRC {X -231.692,Y 157.532,Z -20.000,A 0.015,B 0.000,C -180.000},{X -235.201,Y 159.110,Z -20.000,A 0.015,B 0.000,C 180.000} C_DIS
CIRC {X -257.169,Y 164.183,Z -20.000,A 0.015,B 0.000,C 180.000},{X -278.034,Y 172.730,Z -20.000,A 0.015,B 0.000,C 180.000} C_DIS
CIRC {X -281.479,Y 174.616,Z -20.000,A 0.015,B 0.000,C 180.000},{X -284.783,Y 176.740,Z -20.000,A 0.015,B 0.000,C -180.000} C_DIS
CIRC {X -288.027,Y 178.951,Z -20.000,A 0.015,B 0.000,C 180.000},{X -291.307,Y 181.107,Z -20.000,A 0.015,B 0.000,C -180.000} C_DIS
CIRC {X -293.477,Y 181.188,Z -20.000,A 0.015,B 0.000,C 180.000},{X -294.586,Y 179.321,Z -20.000,A 0.015,B 0.000,C 180.000} C_DIS
LIN {X -294.585,Y 153.807,Z -20.000,A 0.015,B 0.000,C -180.000} C_DIS
CIRC {X -293.488,Y 149.378,Z -20.000,A 0.015,B 0.000,C -180.000},{X -290.451,Y 145.974,Z -20.000,A 0.015,B 0.000,C -180.000} C_DIS
CIRC {X -280.550,Y 138.556,Z -20.000,A 0.015,B -0.000,C -180.000},{X -271.327,Y 130.310,Z -20.000,A 0.015,B 0.000,C -180.000} C_DIS
CIRC {X -262.814,Y 121.336,Z -20.000,A 0.015,B 0.000,C -180.000},{X -255.026,Y 111.726,Z -20.000,A 0.015,B 0.000,C 180.000} C_DIS
CIRC {X -251.145,Y 106.201,Z -20.000,A 0.015,B 0.000,C -180.000},{X -247.601,Y 100.455,Z -20.000,A 0.015,B 0.000,C 180.000} C_DIS
CIRC {X -245.065,Y 95.918,Z -20.000,A 0.015,B 0.000,C 180.000},{X -242.648,Y 91.316,Z -20.000,A 0.015,B 0.000,C -180.000} C_DIS
CIRC {X -240.232,Y 86.715,Z -20.000,A 0.015,B 0.000,C -180.000},{X -237.696,Y 82.178,Z -20.000,A 0.015,B 0.000,C -180.000} C_DIS
CIRC {X -234.591,Y 79.069,Z -20.000,A 0.015,B 0.000,C -180.000},{X -230.347,Y 77.931,Z -20.000,A 0.015,B 0.000,C -180.000} C_DIS
LIN {X -163.189,Y 77.931,Z -20.000,A 0.015,B -0.000,C 180.000} C_DIS
CIRC {X -158.939,Y 79.069,Z -20.000,A 0.015,B 0.000,C 180.000},{X -155.828,Y 82.179,Z -20.000,A 0.015,B 0.000,C 180.000} C_DIS
CIRC {X -153.226,Y 86.816,Z -20.000,A 0.015,B 0.000,C -180.000},{X -150.744,Y 91.519,Z -20.000,A 0.015,B 0.000,C 180.000} C_DIS
CIRC {X -148.261,Y 96.222,Z -20.000,A 0.015,B 0.000,C 180.000},{X -145.659,Y 100.859,Z -20.000,A 0.015,B 0.000,C 180.000} C_DIS
CIRC {X -137.057,Y 113.897,Z -20.000,A 0.015,B 0.000,C -180.000},{X -126.974,Y 125.828,Z -20.000,A 0.015,B 0.000,C -180.000} C_DIS
CIRC {X -115.601,Y 136.530,Z -20.000,A 0.015,B 0.000,C 180.000},{X -103.125,Y 145.922,Z -20.000,A 0.015,B 0.000,C -180.000} C_DIS
CIRC {X -100.042,Y 149.330,Z -20.000,A 0.015,B 0.000,C 180.000},{X -98.927,Y 153.788,Z -20.000,A 0.015,B -0.000,C 180.000} C_DIS
LIN {X -98.928,Y 179.332,Z -20.000,A 0.015,B 0.000,C -180.000} C_DIS
CIRC {X -100.034,Y 181.194,Z -20.000,A 0.015,B 0.000,C 180.000},{X -102.198,Y 181.111,Z -20.000,A 0.015,B 0.000,C 180.000} C_DIS
CIRC {X -109.981,Y 176.308,Z -20.000,A 0.015,B 0.000,C 180.000},{X -117.963,Y 171.846,Z -20.000,A 0.015,B 0.000,C 180.000} C_DIS
CIRC {X -126.223,Y 167.907,Z -20.000,A 0.015,B 0.000,C -180.000},{X -134.792,Y 164.694,Z -20.000,A 0.015,B 0.000,C 180.000} C_DIS
CIRC {X -154.429,Y 159.861,Z -20.000,A 0.015,B 0.000,C -180.000},{X -174.564,Y 157.992,Z -20.000,A 0.015,B 0.000,C -180.000} C_DIS
LIN {X -214.895,Y 157.624,Z -20.000,A 0.015,B 0.000,C 180.000} C_DIS
CIRC {X -225.075,Y 157.996,Z -20.000,A 0.015,B 0.000,C 180.000},{X -235.201,Y 159.110,Z -20.000,A 0.015,B 0.000,C -180.000} C_DIS
CIRC {X -238.609,Y 160.732,Z -20.000,A 0.015,B 0.000,C 180.000},{X -240.518,Y 163.989,Z -20.000,A 0.015,B -0.000,C 180.000} C_DIS
CIRC {X -242.343,Y 167.265,Z -20.000,A 0.015,B 0.000,C 180.000},{X -245.615,Y 169.098,Z -20.000,A 0.015,B 0.000,C 180.000} C_DIS
CIRC {X -260.382,Y 173.552,Z -20.000,A 0.015,B -0.000,C 180.000},{X -274.529,Y 179.697,Z -20.000,A 0.015,B 0.000,C 180.000} C_DIS
CIRC {X -281.079,Y 183.314,Z -20.000,A 0.015,B 0.000,C 180.000},{X -287.330,Y 187.425,Z -20.000,A 0.015,B -0.000,C 180.000} C_DIS
CIRC {X -293.357,Y 191.849,Z -20.000,A 0.015,B -0.000,C -180.000},{X -299.271,Y 196.424,Z -20.000,A 0.015,B -0.000,C 180.000} C_DIS
CIRC {X -301.335,Y 196.654,Z -20.000,A 0.015,B -0.000,C 180.000},{X -302.439,Y 194.895,Z -20.000,A 0.015,B -0.000,C 180.000} C_DIS
LIN {X -302.438,Y 149.182,Z -20.000,A 0.015,B 0.000,C -180.000} C_DIS
CIRC {X -301.341,Y 144.933,Z -20.000,A 0.015,B 0.000,C -180.000},{X -298.326,Y 141.746,Z -20.000,A 0.015,B 0.000,C -180.000} C_DIS
CIRC {X -287.876,Y 134.428,Z -20.000,A 0.015,B 0.000,C 180.000},{X -278.217,Y 126.093,Z -20.000,A 0.015,B 0.000,C 180.000} C_DIS
CIRC {X -269.370,Y 116.909,Z -20.000,A 0.015,B 0.000,C 180.000},{X -261.315,Y 107.023,Z -20.000,A 0.015,B 0.000,C -180.000} C_DIS
CIRC {X -257.703,Y 101.881,Z -20.000,A 0.015,B 0.000,C 180.000},{X -254.405,Y 96.534,Z -20.000,A 0.015,B 0.000,C 180.000} C_DIS
CIRC {X -251.303,Y 91.014,Z -20.000,A 0.015,B -0.000,C 180.000},{X -248.320,Y 85.429,Z -20.000,A 0.015,B 0.000,C -180.000} C_DIS
CIRC {X -245.336,Y 79.844,Z -20.000,A 0.015,B 0.000,C -180.000},{X -242.234,Y 74.325,Z -20.000,A 0.015,B 0.000,C -180.000} C_DIS
CIRC {X -239.129,Y 71.216,Z -20.000,A 0.015,B -0.000,C -180.000},{X -234.885,Y 70.078,Z -20.000,A 0.015,B 0.000,C 180.000} C_DIS
LIN {X -158.657,Y 70.078,Z -20.000,A 0.015,B 0.000,C -180.000} C_DIS
CIRC {X -154.407,Y 71.216,Z -20.000,A 0.015,B -0.000,C 180.000},{X -151.296,Y 74.326,Z -20.000,A 0.015,B 0.000,C -180.000} C_DIS
LIN {X -138.860,Y 96.930,Z -20.000,A 0.015,B -0.000,C 180.000} C_DIS
CIRC {X -130.100,Y 110.064,Z -20.000,A 0.015,B 0.000,C 180.000},{X -119.730,Y 121.970,Z -20.000,A 0.015,B 0.000,C -180.000} C_DIS
CIRC {X -108.013,Y 132.540,Z -20.000,A 0.015,B 0.000,C -180.000},{X -95.187,Y 141.732,Z -20.000,A 0.015,B 0.000,C -180.000} C_DIS
CIRC {X -92.170,Y 144.946,Z -20.000,A 0.015,B -0.000,C 180.000},{X -91.074,Y 149.217,Z -20.000,A 0.015,B -0.000,C 180.000} C_DIS
LIN {X -91.075,Y 194.917,Z -20.000,A 0.015,B 0.000,C 180.000} C_DIS
CIRC {X -92.179,Y 196.681,Z -20.000,A 0.015,B 0.000,C 180.000},{X -94.248,Y 196.458,Z -20.000,A 0.015,B 0.000,C -180.000} C_DIS
CIRC {X -101.574,Y 190.919,Z -20.000,A 0.015,B 0.000,C 180.000},{X -109.109,Y 185.669,Z -20.000,A 0.015,B 0.000,C 180.000} C_DIS
CIRC {X -116.953,Y 180.881,Z -20.000,A 0.015,B -0.000,C -180.000},{X -125.164,Y 176.755,Z -20.000,A 0.015,B 0.000,C -180.000} C_DIS
CIRC {X -146.791,Y 169.399,Z -20.000,A 0.015,B 0.000,C 180.000},{X -169.429,Y 166.337,Z -20.000,A 0.015,B 0.000,C 180.000} C_DIS
LIN {X -214.895,Y 165.478,Z -20.000,A 0.015,B 0.000,C -180.000} C_DIS
CIRC {X -230.361,Y 166.386,Z -20.000,A 0.015,B 0.000,C -180.000},{X -245.615,Y 169.098,Z -20.000,A 0.015,B 0.000,C -180.000} C_DIS
CIRC {X -248.758,Y 170.953,Z -20.000,A 0.015,B 0.000,C -180.000},{X -250.313,Y 174.255,Z -20.000,A 0.015,B 0.000,C 180.000} C_DIS
CIRC {X -251.781,Y 177.570,Z -20.000,A 0.015,B 0.000,C 180.000},{X -254.767,Y 179.626,Z -20.000,A 0.015,B -0.000,C -180.000} C_DIS
CIRC {X -283.101,Y 193.499,Z -20.000,A 0.015,B 0.000,C 180.000},{X -307.013,Y 214.079,Z -20.000,A 0.015,B 0.000,C -180.000} C_DIS
CIRC {X -308.897,Y 214.539,Z -20.000,A 0.015,B 0.000,C -180.000},{X -309.997,Y 212.942,Z -20.000,A 0.015,B 0.000,C -180.000} C_DIS
LIN {X -309.995,Y 144.514,Z -20.000,A 0.015,B 0.000,C -180.000} C_DIS
CIRC {X -308.898,Y 140.443,Z -20.000,A 0.015,B 0.000,C -180.000},{X -305.904,Y 137.475,Z -20.000,A 0.015,B 0.000,C -180.000} C_DIS
CIRC {X -294.916,Y 130.338,Z -20.000,A 0.015,B 0.000,C 180.000},{X -284.832,Y 121.972,Z -20.000,A 0.015,B 0.000,C -180.000} C_DIS
CIRC {X -275.667,Y 112.622,Z -20.000,A 0.015,B 0.000,C 180.000},{X -267.367,Y 102.496,Z -20.000,A 0.015,B 0.000,C -180.000} C_DIS
CIRC {X -264.015,Y 97.724,Z -20.000,A 0.015,B 0.000,C 180.000},{X -260.954,Y 92.760,Z -20.000,A 0.015,B 0.000,C 180.000} C_DIS
LIN {X -246.602,Y 66.767,Z -20.000,A 0.015,B -0.000,C 180.000} C_DIS
CIRC {X -243.497,Y 63.658,Z -20.000,A 0.015,B 0.000,C 180.000},{X -239.253,Y 62.520,Z -20.000,A 0.015,B -0.000,C -180.000} C_DIS
LIN {X -154.295,Y 62.520,Z -20.000,A 0.015,B 0.000,C -180.000} C_DIS
CIRC {X -150.046,Y 63.658,Z -20.000,A 0.015,B 0.000,C -180.000},{X -146.935,Y 66.768,Z -20.000,A 0.015,B -0.000,C 180.000} C_DIS
LIN {X -132.316,Y 93.148,Z -20.000,A 0.015,B -0.000,C -180.000} C_DIS
CIRC {X -123.445,Y 106.360,Z -20.000,A 0.015,B 0.000,C -180.000},{X -112.879,Y 118.262,Z -20.000,A 0.015,B 0.000,C -180.000} C_DIS
CIRC {X -100.855,Y 128.680,Z -20.000,A 0.015,B -0.000,C 180.000},{X -87.606,Y 137.489,Z -20.000,A 0.015,B 0.000,C 180.000} C_DIS
CIRC {X -84.612,Y 140.482,Z -20.000,A 0.015,B 0.000,C -180.000},{X -83.516,Y 144.571,Z -20.000,A 0.015,B -0.000,C 180.000} C_DIS
LIN {X -83.518,Y 212.938,Z -20.000,A 0.015,B 0.000,C 180.000} C_DIS
CIRC {X -84.618,Y 214.535,Z -20.000,A 0.015,B -0.000,C 180.000},{X -86.502,Y 214.075,Z -20.000,A 0.015,B 0.000,C 180.000} C_DIS
CIRC {X -101.262,Y 200.161,Z -20.000,A 0.015,B 0.000,C -180.000},{X -118.197,Y 188.996,Z -20.000,A 0.015,B 0.000,C -180.000} C_DIS
CIRC {X -136.698,Y 180.723,Z -20.000,A 0.015,B 0.000,C -180.000},{X -156.237,Y 175.339,Z -20.000,A 0.015,B -0.000,C -180.000} C_DIS
CIRC {X -170.806,Y 173.281,Z -20.000,A 0.015,B 0.000,C 180.000},{X -185.510,Y 172.770,Z -20.000,A 0.015,B 0.000,C 180.000} C_DIS
LIN {X -214.895,Y 173.035,Z -20.000,A 0.015,B 0.000,C 180.000} C_DIS
CIRC {X -235.102,Y 174.694,Z -20.000,A 0.015,B -0.000,C -180.000},{X -254.767,Y 179.626,Z -20.000,A 0.015,B 0.000,C -180.000} C_DIS
CIRC {X -257.526,Y 181.620,Z -20.000,A 0.015,B 0.000,C 180.000},{X -258.689,Y 184.819,Z -20.000,A 0.015,B 0.000,C 180.000} C_DIS
CIRC {X -259.774,Y 188.021,Z -20.000,A 0.015,B 0.000,C -180.000},{X -262.376,Y 190.181,Z -20.000,A 0.015,B 0.000,C 180.000} C_DIS
CIRC {X -263.778,Y 190.813,Z -20.000,A 0.015,B 0.000,C -180.000},{X -265.172,Y 191.464,Z -20.000,A 0.015,B 0.000,C -180.000} C_DIS
CIRC {X -287.251,Y 205.041,Z -20.000,A 0.015,B 0.000,C -180.000},{X -305.908,Y 223.034,Z -20.000,A 0.015,B -0.000,C 180.000} C_DIS
CIRC {X -308.178,Y 225.948,Z -20.000,A 0.015,B 0.000,C 180.000},{X -310.248,Y 229.008,Z -20.000,A 0.015,B 0.000,C 180.000} C_DIS
CIRC {X -312.235,Y 232.120,Z -20.000,A 0.015,B 0.000,C -180.000},{X -314.265,Y 235.204,Z -20.000,A 0.015,B -0.000,C -180.000} C_DIS
CIRC {X -316.000,Y 235.824,Z -20.000,A 0.015,B -0.000,C 180.000},{X -317.096,Y 234.344,Z -20.000,A 0.015,B 0.000,C 180.000} C_DIS
LIN {X -317.094,Y 140.153,Z -20.000,A 0.015,B 0.000,C -180.000} C_DIS
CIRC {X -315.957,Y 136.079,Z -20.000,A 0.015,B 0.000,C 180.000},{X -312.875,Y 133.181,Z -20.000,A 0.015,B -0.000,C 180.000} C_DIS
CIRC {X -292.126,Y 119.151,Z -20.000,A 0.015,B -0.000,C -180.000},{X -275.010,Y 100.864,Z -20.000,A 0.015,B 0.000,C 180.000} C_DIS
CIRC {X -272.924,Y 98.027,Z -20.000,A 0.015,B -0.000,C 180.000},{X -270.883,Y 95.158,Z -20.000,A 0.015,B -0.000,C -180.000} C_DIS
CIRC {X -268.929,Y 92.228,Z -20.000,A 0.015,B -0.000,C -180.000},{X -267.104,Y 89.216,Z -20.000,A 0.015,B 0.000,C 180.000} C_DIS
LIN {X -250.686,Y 59.638,Z -20.000,A 0.015,B 0.000,C 180.000} C_DIS
CIRC {X -247.604,Y 56.552,Z -20.000,A 0.015,B -0.000,C 180.000},{X -243.390,Y 55.422,Z -20.000,A 0.015,B 0.000,C 180.000} C_DIS
LIN {X -150.139,Y 55.422,Z -20.000,A 0.015,B 0.000,C -180.000} C_DIS
CIRC {X -145.942,Y 56.546,Z -20.000,A 0.015,B -0.000,C 180.000},{X -142.868,Y 59.618,Z -20.000,A 0.015,B 0.000,C -180.000} C_DIS
LIN {X -126.170,Y 89.597,Z -20.000,A 0.015,B 0.000,C 180.000} C_DIS
CIRC {X -106.493,Y 114.663,Z -20.000,A 0.015,B 0.000,C -180.000},{X -80.598,Y 133.237,Z -20.000,A 0.015,B 0.000,C -180.000} C_DIS
CIRC {X -77.544,Y 136.095,Z -20.000,A 0.015,B -0.000,C 180.000},{X -76.417,Y 140.123,Z -20.000,A 0.015,B 0.000,C -180.000} C_DIS
LIN {X -76.420,Y 234.337,Z -20.000,A 0.015,B 0.000,C 180.000} C_DIS
CIRC {X -77.517,Y 235.817,Z -20.000,A 0.015,B 0.000,C 180.000},{X -79.251,Y 235.197,Z -20.000,A 0.015,B 0.000,C -180.000} C_DIS
CIRC {X -84.844,Y 227.285,Z -20.000,A 0.015,B 0.000,C 180.000},{X -90.834,Y 219.670,Z -20.000,A 0.015,B -0.000,C 180.000} C_DIS
CIRC {X -97.420,Y 212.548,Z -20.000,A 0.015,B 0.000,C -180.000},{X -104.734,Y 206.176,Z -20.000,A 0.015,B 0.000,C -180.000} C_DIS
CIRC {X -118.752,Y 196.765,Z -20.000,A 0.015,B 0.000,C 180.000},{X -133.968,Y 189.444,Z -20.000,A 0.015,B 0.000,C 180.000} C_DIS
CIRC {X -150.004,Y 184.198,Z -20.000,A 0.015,B 0.000,C 180.000},{X -166.560,Y 180.939,Z -20.000,A 0.015,B 0.000,C 180.000} C_DIS
CIRC {X -172.575,Y 180.335,Z -20.000,A 0.015,B -0.000,C -180.000},{X -178.617,Y 180.134,Z -20.000,A 0.015,B -0.000,C 180.000} C_DIS
LIN {X -214.895,Y 180.134,Z -20.000,A 0.015,B 0.000,C -180.000} C_DIS
CIRC {X -239.161,Y 182.673,Z -20.000,A 0.015,B -0.000,C 180.000},{X -262.376,Y 190.181,Z -20.000,A 0.015,B 0.000,C -180.000} C_DIS
CIRC {X -264.765,Y 192.255,Z -20.000,A 0.015,B -0.000,C 180.000},{X -265.580,Y 195.311,Z -20.000,A 0.015,B 0.000,C 180.000} C_DIS
CIRC {X -266.324,Y 198.365,Z -20.000,A 0.015,B 0.000,C -180.000},{X -268.559,Y 200.574,Z -20.000,A 0.015,B -0.000,C 180.000} C_DIS
CIRC {X -298.309,Y 224.412,Z -20.000,A 0.015,B 0.000,C 180.000},{X -318.264,Y 256.894,Z -20.000,A 0.015,B 0.000,C 180.000} C_DIS
CIRC {X -321.437,Y 258.630,Z -20.000,A 0.015,B 0.000,C 180.000},{X -323.739,Y 255.842,Z -20.000,A 0.015,B 0.000,C -180.000} C_DIS
LIN {X -323.736,Y 135.887,Z -20.000,A 0.015,B 0.000,C -180.000} C_DIS
CIRC {X -322.643,Y 131.997,Z -20.000,A 0.015,B -0.000,C -180.000},{X -319.683,Y 129.247,Z -20.000,A 0.015,B 0.000,C -180.000} C_DIS
LIN {X -311.689,Y 125.167,Z -20.000,A 0.015,B 0.000,C -180.000} C_DIS
CIRC {X -307.760,Y 122.992,Z -20.000,A 0.015,B -0.000,C -180.000},{X -304.003,Y 120.533,Z -20.000,A 0.015,B 0.000,C 180.000} C_DIS
CIRC {X -296.768,Y 114.825,Z -20.000,A 0.015,B 0.000,C 180.000},{X -290.159,Y 108.402,Z -20.000,A 0.015,B 0.000,C -180.000} C_DIS
CIRC {X -284.078,Y 101.491,Z -20.000,A 0.015,B 0.000,C -180.000},{X -278.370,Y 94.267,Z -20.000,A 0.015,B -0.000,C -180.000} C_DIS
LIN {X -254.451,Y 52.842,Z -20.000,A 0.015,B 0.000,C 180.000} C_DIS
CIRC {X -251.563,Y 49.871,Z -20.000,A 0.015,B 0.000,C 180.000},{X -247.566,Y 48.780,Z -20.000,A 0.015,B 0.000,C -180.000} C_DIS
LIN {X -145.929,Y 48.780,Z -20.000,A 0.015,B 0.000,C 180.000} C_DIS
CIRC {X -141.950,Y 49.871,Z -20.000,A 0.015,B 0.000,C 180.000},{X -139.085,Y 52.840,Z -20.000,A 0.015,B 0.000,C 180.000} C_DIS
LIN {X -119.823,Y 86.739,Z -20.000,A 0.015,B 0.000,C -180.000} C_DIS
CIRC {X -108.496,Y 102.689,Z -20.000,A 0.015,B 0.000,C 180.000},{X -94.666,Y 116.526,Z -20.000,A 0.015,B 0.000,C 180.000} C_DIS
CIRC {X -89.817,Y 120.239,Z -20.000,A 0.015,B 0.000,C -180.000},{X -84.632,Y 123.467,Z -20.000,A 0.015,B 0.000,C 180.000} C_DIS
CIRC {X -79.278,Y 126.391,Z -20.000,A 0.015,B 0.000,C 180.000},{X -73.874,Y 129.223,Z -20.000,A 0.015,B 0.000,C 180.000} C_DIS
CIRC {X -70.881,Y 132.002,Z -20.000,A 0.015,B 0.000,C -180.000},{X -69.775,Y 135.934,Z -20.000,A 0.015,B 0.000,C -180.000} C_DIS
LIN {X -69.778,Y 255.828,Z -20.000,A 0.015,B 0.000,C 180.000} C_DIS
CIRC {X -72.081,Y 258.616,Z -20.000,A 0.015,B -0.000,C 180.000},{X -75.253,Y 256.881,Z -20.000,A 0.015,B 0.000,C 180.000} C_DIS
CIRC {X -102.400,Y 217.039,Z -20.000,A 0.015,B 0.000,C -180.000},{X -143.842,Y 192.405,Z -20.000,A 0.015,B -0.000,C 180.000} C_DIS
CIRC {X -161.304,Y 188.192,Z -20.000,A 0.015,B -0.000,C -180.000},{X -179.211,Y 186.776,Z -20.000,A 0.015,B 0.000,C -180.000} C_DIS
LIN {X -214.895,Y 186.776,Z -20.000,A 0.015,B 0.000,C 180.000} C_DIS
CIRC {X -242.600,Y 190.281,Z -20.000,A 0.015,B 0.000,C 180.000},{X -268.559,Y 200.574,Z -20.000,A 0.015,B 0.000,C 180.000} C_DIS
CIRC {X -271.661,Y 203.783,Z -20.000,A 0.015,B 0.000,C -180.000},{X -272.417,Y 208.181,Z -20.000,A 0.015,B 0.000,C -180.000} C_DIS
CIRC {X -273.026,Y 212.560,Z -20.000,A 0.015,B 0.000,C -180.000},{X -275.778,Y 216.020,Z -20.000,A 0.015,B 0.000,C -180.000} C_DIS
CIRC {X -297.221,Y 237.529,Z -20.000,A 0.015,B 0.000,C -180.000},{X -311.094,Y 264.547,Z -20.000,A 0.015,B 0.000,C 180.000} C_DIS
CIRC {X -313.201,Y 267.422,Z -20.000,A 0.015,B 0.000,C -180.000},{X -316.591,Y 268.518,Z -20.000,A 0.015,B 0.000,C 180.000} C_DIS
LIN {X -329.249,Y 268.518,Z -20.000,A 0.015,B 0.000,C 180.000} C_DIS
CIRC {X -331.974,Y 267.389,Z -20.000,A 0.015,B 0.000,C -180.000},{X -333.102,Y 264.665,Z -20.000,A 0.015,B 0.000,C 180.000} C_DIS
LIN {X -333.098,Y 129.762,Z -20.000,A 0.015,B -0.000,C -180.000} C_DIS
CIRC {X -331.966,Y 125.906,Z -20.000,A 0.015,B 0.000,C 180.000},{X -328.929,Y 123.275,Z -20.000,A 0.015,B 0.000,C -180.000} C_DIS
CIRC {X -319.507,Y 118.553,Z -20.000,A 0.015,B 0.000,C 180.000},{X -310.452,Y 113.160,Z -20.000,A 0.015,B 0.000,C -180.000} C_DIS
CIRC {X -302.012,Y 106.816,Z -20.000,A 0.015,B 0.000,C -180.000},{X -294.554,Y 99.341,Z -20.000,A 0.015,B -0.000,C -180.000} C_DIS
CIRC {X -284.361,Y 86.411,Z -20.000,A 0.015,B -0.000,C -180.000},{X -275.392,Y 72.604,Z -20.000,A 0.015,B 0.000,C 180.000} C_DIS
CIRC {X -267.424,Y 58.209,Z -20.000,A 0.015,B 0.000,C -180.000},{X -260.182,Y 43.436,Z -20.000,A 0.015,B -0.000,C -180.000} C_DIS
CIRC {X -257.635,Y 40.508,Z -20.000,A 0.015,B -0.000,C 180.000},{X -253.910,Y 39.417,Z -20.000,A 0.015,B 0.000,C -180.000} C_DIS
LIN {X -139.560,Y 39.417,Z -20.000,A 0.015,B -0.000,C 180.000} C_DIS
CIRC {X -135.847,Y 40.510,Z -20.000,A 0.015,B 0.000,C 180.000},{X -133.319,Y 43.440,Z -20.000,A 0.015,B 0.000,C 180.000} C_DIS
CIRC {X -132.571,Y 45.105,Z -20.000,A 0.015,B -0.000,C 180.000},{X -131.833,Y 46.774,Z -20.000,A 0.015,B 0.000,C 180.000} C_DIS
CIRC {X -131.055,Y 48.425,Z -20.000,A 0.015,B 0.000,C 180.000},{X -130.186,Y 50.031,Z -20.000,A 0.015,B 0.000,C 180.000} C_DIS
LIN {X -109.602,Y 85.221,Z -20.000,A 0.015,B -0.000,C -180.000} C_DIS
CIRC {X -97.216,Y 101.578,Z -20.000,A 0.015,B 0.000,C -180.000},{X -81.465,Y 114.724,Z -20.000,A 0.015,B 0.000,C 180.000} C_DIS
CIRC {X -77.415,Y 117.184,Z -20.000,A 0.015,B 0.000,C 180.000},{X -73.197,Y 119.345,Z -20.000,A 0.015,B 0.000,C 180.000} C_DIS
CIRC {X -68.900,Y 121.334,Z -20.000,A 0.015,B 0.000,C -180.000},{X -64.587,Y 123.292,Z -20.000,A 0.015,B 0.000,C 180.000} C_DIS
CIRC {X -61.547,Y 125.903,Z -20.000,A 0.015,B 0.000,C -180.000},{X -60.412,Y 129.747,Z -20.000,A 0.015,B 0.000,C 180.000} C_DIS
LIN {X -60.416,Y 264.671,Z -20.000,A 0.015,B 0.000,C -180.000} C_DIS
CIRC {X -61.544,Y 267.396,Z -20.000,A 0.015,B 0.000,C -180.000},{X -64.269,Y 268.524,Z -20.000,A 0.015,B 0.000,C -180.000} C_DIS
LIN {X -76.919,Y 268.524,Z -20.000,A 0.015,B 0.000,C -180.000} C_DIS
CIRC {X -80.310,Y 267.427,Z -20.000,A 0.015,B 0.000,C -180.000},{X -82.416,Y 264.553,Z -20.000,A 0.015,B 0.000,C -180.000} C_DIS
CIRC {X -92.359,Y 243.421,Z -20.000,A 0.015,B -0.000,C 180.000},{X -107.048,Y 225.265,Z -20.000,A 0.015,B -0.000,C 180.000} C_DIS
CIRC {X -125.530,Y 211.019,Z -20.000,A 0.015,B 0.000,C -180.000},{X -146.748,Y 201.305,Z -20.000,A 0.015,B 0.000,C -180.000} C_DIS
CIRC {X -163.470,Y 197.299,Z -20.000,A 0.015,B 0.000,C 180.000},{X -180.618,Y 196.027,Z -20.000,A 0.015,B 0.000,C -180.000} C_DIS
LIN {X -214.895,Y 196.139,Z -20.000,A 0.015,B -0.000,C -180.000} C_DIS
CIRC {X -245.911,Y 200.911,Z -20.000,A 0.015,B -0.000,C 180.000},{X -274.057,Y 214.787,Z -20.000,A 0.015,B -0.000,C 180.000} C_DIS
CIRC {X -274.920,Y 215.399,Z -20.000,A 0.015,B 0.000,C -180.000},{X -275.778,Y 216.020,Z -20.000,A 0.015,B 0.000,C 180.000} C_DIS
CIRC {X -278.633,Y 219.891,Z -20.000,A 0.015,B -0.000,C -180.000},{X -278.775,Y 224.699,Z -20.000,A 0.015,B -0.000,C -180.000} C_DIS
CIRC {X -278.730,Y 229.455,Z -20.000,A 0.015,B 0.000,C -180.000},{X -281.088,Y 233.585,Z -20.000,A 0.015,B 0.000,C 180.000} C_DIS
CIRC {X -283.578,Y 236.180,Z -20.000,A 0.015,B 0.000,C -180.000},{X -285.974,Y 238.862,Z -20.000,A 0.015,B 0.000,C 180.000} C_DIS
CIRC {X -297.046,Y 255.282,Z -20.000,A 0.015,B 0.000,C 180.000},{X -303.969,Y 273.837,Z -20.000,A 0.015,B 0.000,C 180.000} C_DIS
CIRC {X -305.844,Y 276.749,Z -20.000,A 0.015,B -0.000,C 180.000},{X -309.117,Y 277.881,Z -20.000,A 0.015,B -0.000,C -180.000} C_DIS
LIN {X -338.612,Y 277.880,Z -20.000,A 0.015,B 0.000,C -180.000} C_DIS
CIRC {X -341.337,Y 276.752,Z -20.000,A 0.015,B 0.000,C -180.000},{X -342.465,Y 274.027,Z -20.000,A 0.015,B 0.000,C 180.000} C_DIS
LIN {X -342.461,Y 123.085,Z -20.000,A 0.015,B 0.000,C 180.000} C_DIS
CIRC {X -341.372,Y 119.552,Z -20.000,A 0.015,B 0.000,C -180.000},{X -338.484,Y 117.244,Z -20.000,A 0.015,B 0.000,C 180.000} C_DIS
CIRC {X -329.772,Y 113.468,Z -20.000,A 0.015,B 0.000,C 180.000},{X -321.336,Y 109.108,Z -20.000,A 0.015,B -0.000,C 180.000} C_DIS
CIRC {X -313.347,Y 103.953,Z -20.000,A 0.015,B 0.000,C 180.000},{X -306.058,Y 97.848,Z -20.000,A 0.015,B 0.000,C 180.000} C_DIS
CIRC {X -295.385,Y 86.016,Z -20.000,A 0.015,B 0.000,C 180.000},{X -286.666,Y 72.679,Z -20.000,A 0.015,B 0.000,C 180.000} C_DIS
LIN {X -271.096,Y 44.983,Z -20.000,A 0.015,B 0.000,C -180.000} C_DIS
CIRC {X -269.731,Y 42.372,Z -20.000,A 0.015,B -0.000,C 180.000},{X -268.583,Y 39.659,Z -20.000,A 0.015,B 0.000,C 180.000} C_DIS
CIRC {X -267.537,Y 36.908,Z -20.000,A 0.015,B 0.000,C 180.000},{X -266.467,Y 34.165,Z -20.000,A 0.015,B 0.000,C -180.000} C_DIS
CIRC {X -264.078,Y 31.179,Z -20.000,A 0.015,B 0.000,C -180.000},{X -260.424,Y 30.054,Z -20.000,A 0.015,B 0.000,C 180.000} C_DIS
LIN {X -133.097,Y 30.054,Z -20.000,A 0.015,B 0.000,C -180.000} C_DIS
CIRC {X -129.465,Y 31.162,Z -20.000,A 0.015,B 0.000,C -180.000},{X -127.070,Y 34.108,Z -20.000,A 0.015,B 0.000,C -180.000} C_DIS
CIRC {X -125.931,Y 36.970,Z -20.000,A 0.015,B 0.000,C -180.000},{X -124.837,Y 39.850,Z -20.000,A 0.015,B 0.000,C 180.000} C_DIS
CIRC {X -123.644,Y 42.692,Z -20.000,A 0.015,B 0.000,C 180.000},{X -122.215,Y 45.424,Z -20.000,A 0.015,B 0.000,C 180.000} C_DIS
LIN {X -103.065,Y 78.561,Z -20.000,A 0.015,B 0.000,C 180.000} C_DIS
CIRC {X -91.346,Y 94.293,Z -20.000,A 0.015,B 0.000,C 180.000},{X -76.319,Y 106.903,Z -20.000,A 0.015,B 0.000,C -180.000} C_DIS
CIRC {X -71.241,Y 109.967,Z -20.000,A 0.015,B 0.000,C 180.000},{X -65.940,Y 112.625,Z -20.000,A 0.015,B 0.000,C 180.000} C_DIS
CIRC {X -60.513,Y 115.004,Z -20.000,A 0.015,B 0.000,C 180.000},{X -55.026,Y 117.245,Z -20.000,A 0.015,B 0.000,C 180.000} C_DIS
CIRC {X -52.138,Y 119.552,Z -20.000,A 0.015,B 0.000,C 180.000},{X -51.049,Y 123.085,Z -20.000,A 0.015,B 0.000,C 180.000} C_DIS
LIN {X -51.053,Y 274.034,Z -20.000,A 0.015,B 0.000,C 180.000} C_DIS
CIRC {X -52.182,Y 276.759,Z -20.000,A 0.015,B 0.000,C -180.000},{X -54.907,Y 277.887,Z -20.000,A 0.015,B 0.000,C -180.000} C_DIS
LIN {X -84.434,Y 277.886,Z -20.000,A 0.015,B 0.000,C -180.000} C_DIS
CIRC {X -87.694,Y 276.753,Z -20.000,A 0.015,B -0.000,C -180.000},{X -89.549,Y 273.842,Z -20.000,A 0.015,B 0.000,C 180.000} C_DIS
CIRC {X -97.532,Y 252.829,Z -20.000,A 0.015,B 0.000,C -180.000},{X -110.654,Y 234.579,Z -20.000,A 0.015,B 0.000,C -180.000} C_DIS
CIRC {X -127.953,Y 220.248,Z -20.000,A 0.015,B 0.000,C -180.000},{X -148.267,Y 210.658,Z -20.000,A 0.015,B 0.000,C 180.000} C_DIS
CIRC {X -155.688,Y 208.513,Z -20.000,A 0.015,B -0.000,C -180.000},{X -163.238,Y 206.880,Z -20.000,A 0.015,B -0.000,C -180.000} C_DIS
CIRC {X -170.896,Y 205.846,Z -20.000,A 0.015,B 0.000,C -180.000},{X -178.617,Y 205.501,Z -20.000,A 0.015,B -0.000,C -180.000} C_DIS
LIN {X -217.328,Y 205.613,Z -20.000,A 0.015,B -0.000,C -180.000} C_DIS
CIRC {X -236.671,Y 207.961,Z -20.000,A 0.015,B 0.000,C 180.000},{X -254.968,Y 214.660,Z -20.000,A 0.015,B 0.000,C -180.000} C_DIS
CIRC {X -268.791,Y 223.069,Z -20.000,A 0.015,B 0.000,C 180.000},{X -281.088,Y 233.585,Z -20.000,A 0.015,B 0.000,C 180.000} C_DIS
CIRC {X -283.167,Y 237.558,Z -20.000,A 0.015,B -0.000,C 180.000},{X -282.632,Y 242.011,Z -20.000,A 0.015,B 0.000,C 180.000} C_DIS
CIRC {X -281.922,Y 246.385,Z -20.000,A 0.015,B 0.000,C 180.000},{X -283.474,Y 250.536,Z -20.000,A 0.015,B 0.000,C -180.000} C_DIS
CIRC {X -286.105,Y 254.488,Z -20.000,A 0.015,B 0.000,C -180.000},{X -288.496,Y 258.589,Z -20.000,A 0.015,B 0.000,C -180.000} C_DIS
CIRC {X -290.933,Y 263.610,Z -20.000,A 0.015,B -0.000,C 180.000},{X -292.897,Y 268.835,Z -20.000,A 0.015,B 0.000,C 180.000} C_DIS
CIRC {X -294.495,Y 274.179,Z -20.000,A 0.015,B 0.000,C 180.000},{X -295.844,Y 279.591,Z -20.000,A 0.015,B 0.000,C -180.000} C_DIS
CIRC {X -296.033,Y 280.494,Z -20.000,A 0.015,B 0.000,C 180.000},{X -296.193,Y 281.402,Z -20.000,A 0.015,B 0.000,C -180.000} C_DIS
CIRC {X -296.353,Y 282.311,Z -20.000,A 0.015,B 0.000,C 180.000},{X -296.541,Y 283.214,Z -20.000,A 0.015,B 0.000,C 180.000} C_DIS
CIRC {X -298.353,Y 286.112,Z -20.000,A 0.015,B 0.000,C 180.000},{X -301.579,Y 287.244,Z -20.000,A 0.015,B 0.000,C -180.000} C_DIS
LIN {X -347.975,Y 287.243,Z -20.000,A 0.015,B 0.000,C -180.000} C_DIS
CIRC {X -350.699,Y 286.114,Z -20.000,A 0.015,B 0.000,C 180.000},{X -351.828,Y 283.390,Z -20.000,A 0.015,B -0.000,C 180.000} C_DIS
LIN {X -351.823,Y 115.591,Z -20.000,A 0.015,B 0.000,C -180.000} C_DIS
CIRC {X -350.735,Y 112.387,Z -20.000,A 0.015,B 0.000,C -180.000},{X -347.920,Y 110.509,Z -20.000,A 0.015,B 0.000,C -180.000} C_DIS
CIRC {X -334.180,Y 105.445,Z -20.000,A 0.015,B 0.000,C -180.000},{X -321.605,Y 97.942,Z -20.000,A 0.015,B 0.000,C 180.000} C_DIS
CIRC {X -310.468,Y 88.468,Z -20.000,A 0.015,B 0.000,C -180.000},{X -300.863,Y 77.444,Z -20.000,A 0.015,B 0.000,C -180.000} C_DIS
LIN {X -279.074,Y 40.386,Z -20.000,A 0.015,B 0.000,C 180.000} C_DIS
CIRC {X -277.167,Y 36.647,Z -20.000,A 0.015,B 0.000,C -180.000},{X -275.653,Y 32.733,Z -20.000,A 0.015,B 0.000,C -180.000} C_DIS
CIRC {X -274.329,Y 28.756,Z -20.000,A 0.015,B 0.000,C 180.000},{X -272.979,Y 24.788,Z -20.000,A 0.015,B 0.000,C -180.000} C_DIS
CIRC {X -270.765,Y 21.821,Z -20.000,A 0.015,B 0.000,C -180.000},{X -267.239,Y 20.692,Z -20.000,A 0.015,B -0.000,C 180.000} C_DIS
LIN {X -126.273,Y 20.692,Z -20.000,A 0.015,B 0.000,C -180.000} C_DIS
CIRC {X -122.747,Y 21.821,Z -20.000,A 0.015,B 0.000,C -180.000},{X -120.533,Y 24.788,Z -20.000,A 0.015,B -0.000,C 180.000} C_DIS
CIRC {X -119.142,Y 28.867,Z -20.000,A 0.015,B 0.000,C 180.000},{X -117.773,Y 32.954,Z -20.000,A 0.015,B -0.000,C -180.000} C_DIS
CIRC {X -116.207,Y 36.975,Z -20.000,A 0.015,B 0.000,C 180.000},{X -114.241,Y 40.816,Z -20.000,A 0.015,B 0.000,C -180.000} C_DIS
LIN {X -96.108,Y 72.462,Z -20.000,A 0.015,B -0.000,C 180.000} C_DIS
CIRC {X -85.219,Y 87.251,Z -20.000,A 0.015,B -0.000,C 180.000},{X -71.173,Y 99.081,Z -20.000,A 0.015,B 0.000,C 180.000} C_DIS
CIRC {X -58.844,Y 105.833,Z -20.000,A 0.015,B 0.000,C -180.000},{X -45.589,Y 110.510,Z -20.000,A 0.015,B 0.000,C -180.000} C_DIS
CIRC {X -42.775,Y 112.387,Z -20.000,A 0.015,B 0.000,C 180.000},{X -41.687,Y 115.591,Z -20.000,A 0.015,B 0.000,C 180.000} C_DIS
LIN {X -41.691,Y 283.397,Z -20.000,A 0.015,B -0.000,C 180.000} C_DIS
CIRC {X -42.820,Y 286.121,Z -20.000,A 0.015,B 0.000,C 180.000},{X -45.544,Y 287.250,Z -20.000,A 0.015,B 0.000,C -180.000} C_DIS
LIN {X -91.878,Y 287.249,Z -20.000,A 0.015,B 0.000,C 180.000} C_DIS
CIRC {X -95.105,Y 286.127,Z -20.000,A 0.015,B 0.000,C -180.000},{X -96.941,Y 283.245,Z -20.000,A 0.015,B 0.000,C -180.000} C_DIS
LIN {X -99.555,Y 271.964,Z -20.000,A 0.015,B -0.000,C 180.000} C_DIS
CIRC {X -101.221,Y 266.405,Z -20.000,A 0.015,B 0.000,C 180.000},{X -103.636,Y 261.128,Z -20.000,A 0.015,B 0.000,C 180.000} C_DIS
CIRC {X -113.770,Y 246.021,Z -20.000,A 0.015,B 0.000,C -180.000},{X -126.521,Y 233.047,Z -20.000,A 0.015,B 0.000,C 180.000} C_DIS
CIRC {X -141.853,Y 223.129,Z -20.000,A 0.015,B 0.000,C 180.000},{X -159.185,Y 217.383,Z -20.000,A 0.015,B 0.000,C -180.000} C_DIS
CIRC {X -164.006,Y 216.480,Z -20.000,A 0.015,B -0.000,C -180.000},{X -168.840,Y 215.654,Z -20.000,A 0.015,B 0.000,C -180.000} C_DIS
CIRC {X -173.712,Y 215.062,Z -20.000,A 0.015,B -0.000,C -180.000},{X -178.617,Y 214.864,Z -20.000,A 0.015,B -0.000,C -180.000} C_DIS
LIN {X -215.166,Y 214.722,Z -20.000,A 0.015,B -0.000,C -180.000} C_DIS
CIRC {X -233.458,Y 216.755,Z -20.000,A 0.015,B -0.000,C -180.000},{X -250.761,Y 223.024,Z -20.000,A 0.015,B 0.000,C 180.000} C_DIS
CIRC {X -262.069,Y 229.726,Z -20.000,A 0.015,B 0.000,C 180.000},{X -272.347,Y 237.922,Z -20.000,A 0.015,B 0.000,C -180.000} C_DIS
CIRC {X -278.244,Y 243.935,Z -20.000,A 0.015,B 0.000,C 180.000},{X -283.474,Y 250.536,Z -20.000,A 0.015,B 0.000,C 180.000} C_DIS
CIRC {X -284.910,Y 255.004,Z -20.000,A 0.015,B 0.000,C 180.000},{X -283.517,Y 259.486,Z -20.000,A 0.015,B 0.000,C 180.000} C_DIS
CIRC {X -281.916,Y 263.823,Z -20.000,A 0.015,B 0.000,C -180.000},{X -282.625,Y 268.392,Z -20.000,A 0.015,B 0.000,C -180.000} C_DIS
CIRC {X -284.965,Y 274.501,Z -20.000,A 0.015,B 0.000,C -180.000},{X -286.781,Y 280.785,Z -20.000,A 0.015,B 0.000,C -180.000} C_DIS
CIRC {X -287.445,Y 283.763,Z -20.000,A 0.015,B 0.000,C -180.000},{X -287.993,Y 286.765,Z -20.000,A 0.015,B 0.000,C 180.000} C_DIS
CIRC {X -288.446,Y 289.782,Z -20.000,A 0.015,B 0.000,C -180.000},{X -288.825,Y 292.809,Z -20.000,A 0.015,B 0.000,C 180.000} C_DIS
CIRC {X -290.226,Y 295.519,Z -20.000,A 0.015,B 0.000,C 180.000},{X -293.076,Y 296.607,Z -20.000,A 0.015,B 0.000,C -180.000} C_DIS
LIN {X -357.338,Y 296.605,Z -20.000,A 0.015,B -0.000,C 180.000} C_DIS
CIRC {X -360.062,Y 295.476,Z -20.000,A 0.015,B -0.000,C 180.000},{X -361.191,Y 292.752,Z -20.000,A 0.015,B 0.000,C 180.000} C_DIS
LIN {X -361.186,Y 107.461,Z -20.000,A 0.015,B -0.000,C -180.000} C_DIS
CIRC {X -360.100,Y 104.492,Z -20.000,A 0.015,B 0.000,C -180.000},{X -357.356,Y 102.923,Z -20.000,A 0.015,B 0.000,C 180.000} C_DIS
CIRC {X -352.527,Y 101.967,Z -20.000,A 0.015,B -0.000,C 180.000},{X -347.755,Y 100.759,Z -20.000,A 0.015,B 0.000,C -180.000} C_DIS
CIRC {X -343.069,Y 99.243,Z -20.000,A 0.015,B 0.000,C 180.000},{X -338.514,Y 97.371,Z -20.000,A 0.015,B 0.000,C -180.000} C_DIS
CIRC {X -321.291,Y 86.214,Z -20.000,A 0.015,B 0.000,C -180.000},{X -308.026,Y 70.556,Z -20.000,A 0.015,B 0.000,C 180.000} C_DIS
LIN {X -287.167,Y 35.722,Z -20.000,A 0.015,B 0.000,C -180.000} C_DIS
CIRC {X -284.692,Y 30.843,Z -20.000,A 0.015,B 0.000,C 180.000},{X -282.749,Y 25.730,Z -20.000,A 0.015,B 0.000,C -180.000} C_DIS
CIRC {X -281.182,Y 20.496,Z -20.000,A 0.015,B 0.000,C 180.000},{X -279.811,Y 15.207,Z -20.000,A 0.015,B 0.000,C -180.000} C_DIS
CIRC {X -278.027,Y 12.415,Z -20.000,A 0.015,B -0.000,C 180.000},{X -274.897,Y 11.329,Z -20.000,A 0.015,B 0.000,C 180.000} C_DIS
LIN {X -118.669,Y 11.329,Z -20.000,A 0.015,B 0.000,C -180.000} C_DIS
CIRC {X -115.499,Y 12.428,Z -20.000,A 0.015,B -0.000,C 180.000},{X -113.689,Y 15.254,Z -20.000,A 0.015,B 0.000,C -180.000} C_DIS
CIRC {X -109.219,Y 29.197,Z -20.000,A 0.015,B 0.000,C -180.000},{X -102.729,Y 42.322,Z -20.000,A 0.015,B 0.000,C -180.000} C_DIS
LIN {X -87.994,Y 67.534,Z -20.000,A 0.015,B 0.000,C -180.000} C_DIS
CIRC {X -80.731,Y 77.748,Z -20.000,A 0.015,B 0.000,C 180.000},{X -71.685,Y 86.423,Z -20.000,A 0.015,B 0.000,C -180.000} C_DIS
CIRC {X -61.426,Y 93.568,Z -20.000,A 0.015,B 0.000,C 180.000},{X -50.363,Y 99.391,Z -20.000,A 0.015,B 0.000,C -180.000} C_DIS
CIRC {X -46.930,Y 100.701,Z -20.000,A 0.015,B 0.000,C -180.000},{X -43.370,Y 101.608,Z -20.000,A 0.015,B 0.000,C -180.000} C_DIS
CIRC {X -39.765,Y 102.286,Z -20.000,A 0.015,B 0.000,C -180.000},{X -36.153,Y 102.923,Z -20.000,A 0.015,B 0.000,C -180.000} C_DIS
CIRC {X -33.409,Y 104.492,Z -20.000,A 0.015,B 0.000,C 180.000},{X -32.324,Y 107.461,Z -20.000,A 0.015,B 0.000,C 180.000} C_DIS
LIN {X -32.329,Y 292.760,Z -20.000,A 0.015,B 0.000,C -180.000} C_DIS
CIRC {X -33.457,Y 295.484,Z -20.000,A 0.015,B 0.000,C 180.000},{X -36.182,Y 296.613,Z -20.000,A 0.015,B 0.000,C -180.000} C_DIS
LIN {X -100.470,Y 296.611,Z -20.000,A 0.015,B -0.000,C 180.000} C_DIS
CIRC {X -103.304,Y 295.523,Z -20.000,A 0.015,B 0.000,C -180.000},{X -104.682,Y 292.818,Z -20.000,A 0.015,B 0.000,C -180.000} C_DIS
CIRC {X -105.792,Y 285.113,Z -20.000,A 0.015,B -0.000,C 180.000},{X -107.494,Y 277.517,Z -20.000,A 0.015,B 0.000,C 180.000} C_DIS
CIRC {X -109.935,Y 270.117,Z -20.000,A 0.015,B -0.000,C 180.000},{X -113.242,Y 263.061,Z -20.000,A 0.015,B 0.000,C 180.000} C_DIS
CIRC {X -122.893,Y 249.423,Z -20.000,A 0.015,B -0.000,C 180.000},{X -135.462,Y 238.416,Z -20.000,A 0.015,B -0.000,C -180.000} C_DIS
CIRC {X -150.104,Y 230.430,Z -20.000,A 0.015,B 0.000,C 180.000},{X -166.061,Y 225.578,Z -20.000,A 0.015,B 0.000,C 180.000} C_DIS
CIRC {X -178.199,Y 223.935,Z -20.000,A 0.015,B 0.000,C 180.000},{X -190.445,Y 223.723,Z -20.000,A 0.015,B 0.000,C 180.000} C_DIS
CIRC {X -202.668,Y 224.100,Z -20.000,A 0.015,B 0.000,C 180.000},{X -214.895,Y 224.226,Z -20.000,A 0.015,B 0.000,C 180.000} C_DIS
CIRC {X -231.101,Y 226.034,Z -20.000,A 0.015,B 0.000,C -180.000},{X -246.511,Y 231.368,Z -20.000,A 0.015,B 0.000,C 180.000} C_DIS
CIRC {X -260.390,Y 239.916,Z -20.000,A 0.015,B 0.000,C -180.000},{X -272.121,Y 251.235,Z -20.000,A 0.015,B 0.000,C -180.000} C_DIS
CIRC {X -277.054,Y 257.929,Z -20.000,A 0.015,B 0.000,C 180.000},{X -281.144,Y 265.170,Z -20.000,A 0.015,B -0.000,C 180.000} C_DIS
CIRC {X -281.903,Y 266.773,Z -20.000,A 0.015,B 0.000,C 180.000},{X -282.625,Y 268.392,Z -20.000,A 0.015,B -0.000,C -180.000} C_DIS
CIRC {X -283.081,Y 272.719,Z -20.000,A 0.015,B -0.000,C -180.000},{X -280.991,Y 276.536,Z -20.000,A 0.015,B 0.000,C 180.000} C_DIS
CIRC {X -278.740,Y 280.184,Z -20.000,A 0.015,B 0.000,C 180.000},{X -278.522,Y 284.466,Z -20.000,A 0.015,B 0.000,C -180.000} C_DIS
CIRC {X -279.666,Y 293.363,Z -20.000,A 0.015,B 0.000,C -180.000},{X -279.514,Y 302.332,Z -20.000,A 0.015,B 0.000,C 180.000} C_DIS
CIRC {X -280.376,Y 304.884,Z -20.000,A 0.015,B 0.000,C 180.000},{X -282.840,Y 305.969,Z -20.000,A 0.015,B 0.000,C 180.000} C_DIS
LIN {X -366.701,Y 305.967,Z -20.000,A 0.015,B 0.000,C 180.000} C_DIS
CIRC {X -369.425,Y 304.839,Z -20.000,A 0.015,B 0.000,C -180.000},{X -370.554,Y 302.114,Z -20.000,A 0.015,B 0.000,C -180.000} C_DIS
LIN {X -370.548,Y 98.687,Z -20.000,A 0.015,B 0.000,C 180.000} C_DIS
CIRC {X -369.456,Y 95.868,Z -20.000,A 0.015,B 0.000,C 180.000},{X -366.749,Y 94.523,Z -20.000,A 0.015,B 0.000,C 180.000} C_DIS
CIRC {X -361.672,Y 94.040,Z -20.000,A 0.015,B 0.000,C 180.000},{X -356.597,Y 93.525,Z -20.000,A 0.015,B -0.000,C -180.000} C_DIS
CIRC {X -351.567,Y 92.583,Z -20.000,A 0.015,B 0.000,C -180.000},{X -346.756,Y 90.842,Z -20.000,A 0.015,B 0.000,C 180.000} C_DIS
CIRC {X -336.966,Y 85.636,Z -20.000,A 0.015,B 0.000,C -180.000},{X -327.876,Y 79.287,Z -20.000,A 0.015,B 0.000,C 180.000} C_DIS
CIRC {X -319.854,Y 71.592,Z -20.000,A 0.015,B 0.000,C -180.000},{X -313.420,Y 62.527,Z -20.000,A 0.015,B 0.000,C -180.000} C_DIS
LIN {X -295.280,Y 31.047,Z -20.000,A 0.015,B 0.000,C -180.000} C_DIS
CIRC {X -292.322,Y 25.099,Z -20.000,A 0.015,B 0.000,C 180.000},{X -290.115,Y 18.834,Z -20.000,A 0.015,B 0.000,C 180.000} C_DIS
CIRC {X -288.591,Y 12.375,Z -20.000,A 0.015,B 0.000,C 180.000},{X -287.662,Y 5.804,Z -20.000,A 0.015,B 0.000,C -180.000} C_DIS
CIRC {X -286.294,Y 3.069,Z -20.000,A 0.015,B -0.000,C 180.000},{X -283.443,Y 1.966,Z -20.000,A 0.015,B -0.000,C 180.000} C_DIS
LIN {X -110.095,Y 1.966,Z -20.000,A 0.015,B 0.000,C 180.000} C_DIS
CIRC {X -107.205,Y 3.081,Z -20.000,A 0.015,B 0.000,C -180.000},{X -105.812,Y 5.848,Z -20.000,A 0.015,B 0.000,C -180.000} C_DIS
CIRC {X -104.849,Y 12.513,Z -20.000,A 0.015,B 0.000,C -180.000},{X -103.290,Y 19.064,Z -20.000,A 0.015,B 0.000,C 180.000} C_DIS
CIRC {X -101.042,Y 25.418,Z -20.000,A 0.015,B 0.000,C 180.000},{X -98.034,Y 31.450,Z -20.000,A 0.015,B 0.000,C -180.000} C_DIS
LIN {X -75.510,Y 69.093,Z -20.000,A 0.015,B -0.000,C -180.000} C_DIS
CIRC {X -67.372,Y 77.949,Z -20.000,A 0.015,B -0.000,C -180.000},{X -57.742,Y 85.152,Z -20.000,A 0.015,B 0.000,C 180.000} C_DIS
CIRC {X -46.968,Y 90.488,Z -20.000,A 0.015,B 0.000,C -180.000},{X -35.415,Y 93.815,Z -20.000,A 0.015,B 0.000,C 180.000} C_DIS
CIRC {X -33.277,Y 94.133,Z -20.000,A 0.015,B -0.000,C -180.000},{X -31.120,Y 94.267,Z -20.000,A 0.015,B -0.000,C 180.000} C_DIS
CIRC {X -28.962,Y 94.345,Z -20.000,A 0.015,B 0.000,C 180.000},{X -26.808,Y 94.496,Z -20.000,A 0.015,B 0.000,C 180.000} C_DIS
CIRC {X -24.068,Y 95.847,Z -20.000,A 0.015,B -0.000,C -180.000},{X -22.961,Y 98.694,Z -20.000,A 0.015,B 0.000,C 180.000} C_DIS
LIN {X -22.966,Y 302.123,Z -20.000,A 0.015,B 0.000,C 180.000} C_DIS
CIRC {X -24.095,Y 304.847,Z -20.000,A 0.015,B 0.000,C 180.000},{X -26.819,Y 305.976,Z -20.000,A 0.015,B -0.000,C 180.000} C_DIS
LIN {X -110.710,Y 305.974,Z -20.000,A 0.015,B 0.000,C -180.000} C_DIS
CIRC {X -113.157,Y 304.881,Z -20.000,A 0.015,B -0.000,C -180.000},{X -113.976,Y 302.329,Z -20.000,A 0.015,B 0.000,C 180.000} C_DIS
CIRC {X -114.354,Y 286.968,Z -20.000,A 0.015,B -0.000,C 180.000},{X -118.777,Y 272.251,Z -20.000,A 0.015,B 0.000,C -180.000} C_DIS
CIRC {X -126.748,Y 259.144,Z -20.000,A 0.015,B 0.000,C -180.000},{X -137.619,Y 248.320,Z -20.000,A 0.015,B -0.000,C 180.000} C_DIS
CIRC {X -145.792,Y 242.877,Z -20.000,A 0.015,B 0.000,C 180.000},{X -154.687,Y 238.721,Z -20.000,A 0.015,B 0.000,C 180.000} C_DIS
CIRC {X -164.043,Y 235.777,Z -20.000,A 0.015,B -0.000,C 180.000},{X -173.672,Y 233.919,Z -20.000,A 0.015,B -0.000,C -180.000} C_DIS
LIN {X -214.895,Y 233.589,Z -20.000,A 0.015,B 0.000,C 180.000} C_DIS
CIRC {X -240.670,Y 238.831,Z -20.000,A 0.015,B -0.000,C 180.000},{X -262.350,Y 253.724,Z -20.000,A 0.015,B 0.000,C -180.000} C_DIS
CIRC {X -272.633,Y 267.939,Z -20.000,A 0.015,B 0.000,C 180.000},{X -278.522,Y 284.466,Z -20.000,A 0.015,B -0.000,C -180.000} C_DIS
CIRC {X -278.092,Y 288.833,Z -20.000,A 0.015,B 0.000,C 180.000},{X -275.281,Y 292.203,Z -20.000,A 0.015,B 0.000,C -180.000} C_DIS
CIRC {X -272.308,Y 295.324,Z -20.000,A 0.015,B -0.000,C -180.000},{X -271.049,Y 299.446,Z -20.000,A 0.015,B -0.000,C 180.000} C_DIS
LIN {X -270.979,Y 300.380,Z -20.000,A 0.015,B 0.000,C -180.000} C_DIS
CIRC {X -270.645,Y 303.134,Z -20.000,A 0.015,B -0.000,C -180.000},{X -270.124,Y 305.858,Z -20.000,A 0.015,B -0.000,C -180.000} C_DIS
CIRC {X -269.559,Y 308.572,Z -20.000,A 0.015,B 0.000,C -180.000},{X -269.091,Y 311.305,Z -20.000,A 0.015,B 0.000,C 180.000} C_DIS
CIRC {X -269.826,Y 313.873,Z -20.000,A 0.015,B 0.000,C -180.000},{X -272.253,Y 314.988,Z -20.000,A 0.015,B 0.000,C -180.000} C_DIS
LIN {X -375.719,Y 314.985,Z -20.000,A 0.015,B 0.000,C 180.000} C_DIS
CIRC {X -378.443,Y 313.856,Z -20.000,A 0.015,B -0.000,C 180.000},{X -379.572,Y 311.132,Z -20.000,A 0.015,B 0.000,C 180.000} C_DIS
LIN {X -379.566,Y 88.792,Z -20.000,A 0.015,B -0.000,C 180.000} C_DIS
CIRC {X -378.491,Y 86.358,Z -20.000,A 0.015,B -0.000,C -180.000},{X -375.969,Y 85.512,Z -20.000,A 0.015,B 0.000,C 180.000} C_DIS
CIRC {X -365.499,Y 85.562,Z -20.000,A 0.015,B 0.000,C 180.000},{X -355.180,Y 83.795,Z -20.000,A 0.015,B 0.000,C -180.000} C_DIS
CIRC {X -345.330,Y 80.237,Z -20.000,A 0.015,B 0.000,C 180.000},{X -336.276,Y 74.975,Z -20.000,A 0.015,B 0.000,C -180.000} C_DIS
CIRC {X -332.494,Y 71.921,Z -20.000,A 0.015,B 0.000,C 180.000},{X -329.125,Y 68.417,Z -20.000,A 0.015,B 0.000,C -180.000} C_DIS
CIRC {X -326.045,Y 64.669,Z -20.000,A 0.015,B 0.000,C 180.000},{X -323.080,Y 60.828,Z -20.000,A 0.015,B 0.000,C 180.000} C_DIS
LIN {X -303.093,Y 26.545,Z -20.000,A 0.015,B 0.000,C 180.000} C_DIS
CIRC {X -300.359,Y 20.995,Z -20.000,A 0.015,B -0.000,C -180.000},{X -298.367,Y 15.139,Z -20.000,A 0.015,B 0.000,C 180.000} C_DIS
CIRC {X -297.043,Y 9.103,Z -20.000,A 0.015,B 0.000,C -180.000},{X -296.291,Y 2.969,Z -20.000,A 0.015,B 0.000,C -180.000} C_DIS
CIRC {X -296.245,Y 1.411,Z -20.000,A 0.015,B 0.000,C 180.000},{X -296.341,Y -0.145,Z -20.000,A 0.015,B 0.000,C 180.000} C_DIS
CIRC {X -296.488,Y -1.695,Z -20.000,A 0.015,B 0.000,C -180.000},{X -296.596,Y -3.248,Z -20.000,A 0.015,B 0.000,C 180.000} C_DIS
CIRC {X -295.618,Y -5.924,Z -20.000,A 0.015,B 0.000,C 180.000},{X -293.002,Y -7.051,Z -20.000,A 0.015,B 0.000,C 180.000} C_DIS
LIN {X -100.510,Y -7.051,Z -20.000,A 0.015,B 0.000,C 180.000} C_DIS
CIRC {X -97.894,Y -5.924,Z -20.000,A 0.015,B -0.000,C -180.000},{X -96.916,Y -3.248,Z -20.000,A 0.015,B 0.000,C 180.000} C_DIS
CIRC {X -97.075,Y 1.010,Z -20.000,A 0.015,B 0.000,C -180.000},{X -97.070,Y 5.271,Z -20.000,A 0.015,B 0.000,C 180.000} C_DIS
CIRC {X -96.652,Y 9.524,Z -20.000,A 0.015,B -0.000,C -180.000},{X -95.581,Y 13.661,Z -20.000,A 0.015,B 0.000,C 180.000} C_DIS
CIRC {X -94.409,Y 17.047,Z -20.000,A 0.015,B 0.000,C 180.000},{X -93.224,Y 20.428,Z -20.000,A 0.015,B 0.000,C -180.000} C_DIS
CIRC {X -91.875,Y 23.752,Z -20.000,A 0.015,B 0.000,C -180.000},{X -90.226,Y 26.938,Z -20.000,A 0.015,B 0.000,C -180.000} C_DIS
LIN {X -68.333,Y 63.633,Z -20.000,A 0.015,B 0.000,C -180.000} C_DIS
CIRC {X -53.019,Y 77.585,Z -20.000,A 0.015,B -0.000,C 180.000},{X -33.750,Y 85.193,Z -20.000,A 0.015,B -0.000,C 180.000} C_DIS
CIRC {X -29.721,Y 85.763,Z -20.000,A 0.015,B 0.000,C 180.000},{X -25.656,Y 85.926,Z -20.000,A 0.015,B 0.000,C 180.000} C_DIS
CIRC {X -21.593,Y 85.802,Z -20.000,A 0.015,B 0.000,C -180.000},{X -17.539,Y 85.512,Z -20.000,A 0.015,B 0.000,C -180.000} C_DIS
CIRC {X -15.017,Y 86.358,Z -20.000,A 0.015,B 0.000,C 180.000},{X -13.943,Y 88.791,Z -20.000,A 0.015,B 0.000,C -180.000} C_DIS
LIN {X -13.949,Y 311.141,Z -20.000,A 0.015,B 0.000,C 180.000} C_DIS
CIRC {X -15.077,Y 313.865,Z -20.000,A 0.015,B 0.000,C 180.000},{X -17.802,Y 314.994,Z -20.000,A 0.015,B 0.000,C 180.000} C_DIS
LIN {X -121.257,Y 314.991,Z -20.000,A 0.015,B 0.000,C 180.000} C_DIS
CIRC {X -123.666,Y 313.888,Z -20.000,A 0.015,B 0.000,C -180.000},{X -124.404,Y 311.343,Z -20.000,A 0.015,B -0.000,C 180.000} C_DIS
CIRC {X -123.617,Y 306.314,Z -20.000,A 0.015,B 0.000,C 180.000},{X -122.752,Y 301.298,Z -20.000,A 0.015,B 0.000,C -180.000} C_DIS
CIRC {X -122.365,Y 296.195,Z -20.000,A 0.015,B 0.000,C 180.000},{X -123.028,Y 291.121,Z -20.000,A 0.015,B -0.000,C 180.000} C_DIS
CIRC {X -124.468,Y 285.354,Z -20.000,A 0.015,B 0.000,C -180.000},{X -126.044,Y 279.623,Z -20.000,A 0.015,B 0.000,C 180.000} C_DIS
CIRC {X -128.174,Y 274.052,Z -20.000,A 0.015,B 0.000,C -180.000},{X -131.217,Y 268.921,Z -20.000,A 0.015,B 0.000,C 180.000} C_DIS
CIRC {X -137.046,Y 261.675,Z -20.000,A 0.015,B 0.000,C 180.000},{X -143.662,Y 255.140,Z -20.000,A 0.015,B -0.000,C 180.000} C_DIS
CIRC {X -151.255,Y 249.713,Z -20.000,A 0.015,B -0.000,C -180.000},{X -159.786,Y 245.931,Z -20.000,A 0.015,B 0.000,C 180.000} C_DIS
CIRC {X -164.391,Y 244.583,Z -20.000,A 0.015,B 0.000,C -180.000},{X -169.070,Y 243.524,Z -20.000,A 0.015,B 0.000,C -180.000} C_DIS
CIRC {X -173.821,Y 242.837,Z -20.000,A 0.015,B 0.000,C 180.000},{X -178.617,Y 242.607,Z -20.000,A 0.015,B 0.000,C -180.000} C_DIS
LIN {X -218.640,Y 242.857,Z -20.000,A 0.015,B 0.000,C 180.000} C_DIS
CIRC {X -230.232,Y 245.340,Z -20.000,A 0.015,B 0.000,C 180.000},{X -241.302,Y 249.584,Z -20.000,A 0.015,B 0.000,C -180.000} C_DIS
CIRC {X -251.325,Y 256.031,Z -20.000,A 0.015,B 0.000,C -180.000},{X -259.388,Y 264.807,Z -20.000,A 0.015,B -0.000,C -180.000} C_DIS
CIRC {X -264.385,Y 272.907,Z -20.000,A 0.015,B -0.000,C 180.000},{X -268.334,Y 281.567,Z -20.000,A 0.015,B 0.000,C -180.000} C_DIS
CIRC {X -270.655,Y 290.360,Z -20.000,A 0.015,B 0.000,C 180.000},{X -271.049,Y 299.446,Z -20.000,A 0.015,B 0.000,C -180.000} C_DIS
CIRC {X -269.563,Y 303.394,Z -20.000,A 0.015,B 0.000,C 180.000},{X -266.126,Y 305.840,Z -20.000,A 0.015,B 0.000,C 180.000} C_DIS
CIRC {X -262.611,Y 308.051,Z -20.000,A 0.015,B 0.000,C 180.000},{X -260.505,Y 311.631,Z -20.000,A 0.015,B 0.000,C -180.000} C_DIS
CIRC {X -258.911,Y 316.069,Z -20.000,A 0.015,B 0.000,C -180.000},{X -256.868,Y 320.320,Z -20.000,A 0.015,B 0.000,C 180.000} C_DIS
CIRC {X -256.909,Y 322.577,Z -20.000,A 0.015,B 0.000,C -180.000},{X -258.870,Y 323.693,Z -20.000,A 0.015,B 0.000,C 180.000} C_DIS
LIN {X -384.425,Y 323.690,Z -20.000,A 0.015,B 0.000,C -180.000} C_DIS
CIRC {X -387.149,Y 322.562,Z -20.000,A 0.015,B 0.000,C -180.000},{X -388.277,Y 319.837,Z -20.000,A 0.015,B 0.000,C -180.000} C_DIS
LIN {X -388.271,Y 77.067,Z -20.000,A 0.015,B 0.000,C 180.000} C_DIS
CIRC {X -387.149,Y 74.831,Z -20.000,A 0.015,B -0.000,C -180.000},{X -384.685,Y 74.394,Z -20.000,A 0.015,B 0.000,C 180.000} C_DIS
CIRC {X -380.779,Y 75.543,Z -20.000,A 0.015,B 0.000,C -180.000},{X -376.865,Y 76.666,Z -20.000,A 0.015,B -0.000,C 180.000} C_DIS
CIRC {X -372.844,Y 77.416,Z -20.000,A 0.015,B -0.000,C -180.000},{X -368.755,Y 77.417,Z -20.000,A 0.015,B 0.000,C -180.000} C_DIS
CIRC {X -359.822,Y 76.012,Z -20.000,A 0.015,B -0.000,C 180.000},{X -351.143,Y 73.476,Z -20.000,A 0.015,B 0.000,C -180.000} C_DIS
CIRC {X -343.056,Y 69.310,Z -20.000,A 0.015,B 0.000,C 180.000},{X -336.278,Y 63.241,Z -20.000,A 0.015,B 0.000,C 180.000} C_DIS
LIN {X -332.333,Y 58.681,Z -20.000,A 0.015,B 0.000,C 180.000} C_DIS
CIRC {X -330.435,Y 56.264,Z -20.000,A 0.015,B 0.000,C -180.000},{X -328.776,Y 53.678,Z -20.000,A 0.015,B 0.000,C 180.000} C_DIS
LIN {X -310.636,Y 22.198,Z -20.000,A 0.015,B 0.000,C -180.000} C_DIS
CIRC {X -307.030,Y 14.065,Z -20.000,A 0.015,B 0.000,C -180.000},{X -305.208,Y 5.357,Z -20.000,A 0.015,B 0.000,C -180.000} C_DIS
CIRC {X -305.026,Y -3.517,Z -20.000,A 0.015,B 0.000,C -180.000},{X -306.263,Y -12.306,Z -20.000,A 0.015,B 0.000,C 180.000} C_DIS
CIRC {X -305.710,Y -14.695,Z -20.000,A 0.015,B 0.000,C -180.000},{X -303.499,Y -15.757,Z -20.000,A 0.015,B 0.000,C 180.000} C_DIS
LIN {X -90.025,Y -15.757,Z -20.000,A 0.015,B -0.000,C 180.000} C_DIS
CIRC {X -87.787,Y -14.671,Z -20.000,A 0.015,B -0.000,C 180.000},{X -87.255,Y -12.241,Z -20.000,A 0.015,B 0.000,C 180.000} C_DIS
CIRC {X -88.254,Y -7.092,Z -20.000,A 0.015,B 0.000,C -180.000},{X -88.790,Y -1.874,Z -20.000,A 0.015,B 0.000,C 180.000} C_DIS
CIRC {X -88.740,Y 3.378,Z -20.000,A 0.015,B 0.000,C 180.000},{X -87.989,Y 8.576,Z -20.000,A 0.015,B 0.000,C -180.000} C_DIS
CIRC {X -87.193,Y 11.636,Z -20.000,A 0.015,B 0.000,C 180.000},{X -86.131,Y 14.613,Z -20.000,A 0.015,B 0.000,C -180.000} C_DIS
LIN {X -83.862,Y 20.186,Z -20.000,A 0.015,B -0.000,C -180.000} C_DIS
LIN {X -64.543,Y 53.982,Z -20.000,A 0.015,B 0.000,C 180.000} C_DIS
CIRC {X -59.675,Y 60.728,Z -20.000,A 0.015,B -0.000,C -180.000},{X -53.553,Y 66.360,Z -20.000,A 0.015,B 0.000,C 180.000} C_DIS
CIRC {X -46.655,Y 70.956,Z -20.000,A 0.015,B 0.000,C 180.000},{X -39.293,Y 74.766,Z -20.000,A 0.015,B 0.000,C 180.000} C_DIS
CIRC {X -34.525,Y 76.401,Z -20.000,A 0.015,B -0.000,C -180.000},{X -29.539,Y 77.136,Z -20.000,A 0.015,B 0.000,C -180.000} C_DIS
CIRC {X -24.522,Y 77.303,Z -20.000,A 0.015,B 0.000,C -180.000},{X -19.502,Y 77.259,Z -20.000,A 0.015,B 0.000,C -180.000} C_DIS
CIRC {X -16.738,Y 76.941,Z -20.000,A 0.015,B 0.000,C 180.000},{X -14.065,Y 76.165,Z -20.000,A 0.015,B 0.000,C 180.000} C_DIS
CIRC {X -11.459,Y 75.218,Z -20.000,A 0.015,B 0.000,C 180.000},{X -8.819,Y 74.369,Z -20.000,A 0.015,B 0.000,C -180.000} C_DIS
CIRC {X -6.359,Y 74.799,Z -20.000,A 0.015,B -0.000,C -180.000},{X -5.237,Y 77.030,Z -20.000,A 0.015,B 0.000,C 180.000} C_DIS
LIN {X -5.244,Y 319.846,Z -20.000,A 0.015,B 0.000,C -180.000} C_DIS
CIRC {X -6.372,Y 322.571,Z -20.000,A 0.015,B 0.000,C 180.000},{X -9.097,Y 323.699,Z -20.000,A 0.015,B 0.000,C 180.000} C_DIS
LIN {X -134.651,Y 323.696,Z -20.000,A 0.015,B 0.000,C 180.000} C_DIS
CIRC {X -136.613,Y 322.580,Z -20.000,A 0.015,B -0.000,C 180.000},{X -136.655,Y 320.322,Z -20.000,A 0.015,B -0.000,C 180.000} C_DIS
CIRC {X -134.114,Y 314.917,Z -20.000,A 0.015,B 0.000,C 180.000},{X -132.230,Y 309.250,Z -20.000,A 0.015,B -0.000,C -180.000} C_DIS
CIRC {X -131.135,Y 303.371,Z -20.000,A 0.015,B 0.000,C 180.000},{X -130.962,Y 297.394,Z -20.000,A 0.015,B 0.000,C -180.000} C_DIS
CIRC {X -135.195,Y 279.730,Z -20.000,A 0.015,B 0.000,C 180.000},{X -145.573,Y 264.822,Z -20.000,A 0.015,B 0.000,C 180.000} C_DIS
CIRC {X -160.767,Y 254.820,Z -20.000,A 0.015,B -0.000,C -180.000},{X -178.617,Y 251.312,Z -20.000,A 0.015,B 0.000,C -180.000} C_DIS
LIN {X -221.109,Y 251.972,Z -20.000,A 0.015,B 0.000,C -180.000} C_DIS
CIRC {X -242.009,Y 260.054,Z -20.000,A 0.015,B 0.000,C 180.000},{X -256.965,Y 276.741,Z -20.000,A 0.015,B -0.000,C 180.000} C_DIS
CIRC {X -262.218,Y 293.833,Z -20.000,A 0.015,B 0.000,C 180.000},{X -260.505,Y 311.631,Z -20.000,A 0.015,B 0.000,C 180.000} C_DIS
CIRC {X -258.358,Y 314.872,Z -20.000,A 0.015,B -0.000,C 180.000},{X -254.780,Y 316.394,Z -20.000,A 0.015,B -0.000,C 180.000} C_DIS
CIRC {X -251.168,Y 317.607,Z -20.000,A 0.015,B -0.000,C 180.000},{X -248.384,Y 320.208,Z -20.000,A 0.015,B -0.000,C 180.000} C_DIS
CIRC {X -246.158,Y 323.470,Z -20.000,A 0.015,B 0.000,C -180.000},{X -243.974,Y 326.761,Z -20.000,A 0.015,B -0.000,C -180.000} C_DIS
CIRC {X -243.570,Y 327.316,Z -20.000,A 0.015,B 0.000,C -180.000},{X -243.113,Y 327.827,Z -20.000,A 0.015,B 0.000,C 180.000} C_DIS
CIRC {X -242.628,Y 328.312,Z -20.000,A 0.015,B 0.000,C -180.000},{X -242.138,Y 328.790,Z -20.000,A 0.015,B 0.000,C 180.000} C_DIS
CIRC {X -241.726,Y 330.729,Z -20.000,A 0.015,B 0.000,C -180.000},{X -243.370,Y 331.838,Z -20.000,A 0.015,B 0.000,C 180.000} C_DIS
LIN {X -392.569,Y 331.834,Z -20.000,A 0.015,B -0.000,C 180.000} C_DIS
CIRC {X -395.293,Y 330.706,Z -20.000,A 0.015,B 0.000,C -180.000},{X -396.422,Y 327.981,Z -20.000,A 0.015,B 0.000,C 180.000} C_DIS
LIN {X -396.415,Y 62.514,Z -20.000,A 0.015,B -0.000,C 180.000} C_DIS
CIRC {X -395.303,Y 60.743,Z -20.000,A 0.015,B 0.000,C 180.000},{X -393.225,Y 60.976,Z -20.000,A 0.015,B 0.000,C -180.000} C_DIS
CIRC {X -391.474,Y 62.375,Z -20.000,A 0.015,B 0.000,C -180.000},{X -389.729,Y 63.780,Z -20.000,A 0.015,B 0.000,C -180.000} C_DIS
CIRC {X -387.848,Y 65.017,Z -20.000,A 0.015,B 0.000,C 180.000},{X -385.763,Y 65.866,Z -20.000,A 0.015,B 0.000,C 180.000} C_DIS
CIRC {X -381.769,Y 67.091,Z -20.000,A 0.015,B -0.000,C -180.000},{X -377.796,Y 68.382,Z -20.000,A 0.015,B 0.000,C -180.000} C_DIS
CIRC {X -373.697,Y 69.294,Z -20.000,A 0.015,B -0.000,C 180.000},{X -369.497,Y 69.344,Z -20.000,A 0.015,B 0.000,C -180.000} C_DIS
CIRC {X -359.590,Y 67.424,Z -20.000,A 0.015,B -0.000,C -180.000},{X -350.260,Y 63.580,Z -20.000,A 0.015,B 0.000,C 180.000} C_DIS
CIRC {X -342.066,Y 57.608,Z -20.000,A 0.015,B 0.000,C -180.000},{X -335.832,Y 49.611,Z -20.000,A 0.015,B 0.000,C -180.000} C_DIS
LIN {X -317.692,Y 18.132,Z -20.000,A 0.015,B -0.000,C 180.000} C_DIS
CIRC {X -314.814,Y 11.596,Z -20.000,A 0.015,B 0.000,C 180.000},{X -313.405,Y 4.595,Z -20.000,A 0.015,B 0.000,C 180.000} C_DIS
CIRC {X -313.149,Y -2.510,Z -20.000,A 0.015,B -0.000,C -180.000},{X -313.670,Y -9.602,Z -20.000,A 0.015,B 0.000,C -180.000} C_DIS
CIRC {X -314.335,Y -12.554,Z -20.000,A 0.015,B -0.000,C 180.000},{X -315.539,Y -15.330,Z -20.000,A 0.015,B 0.000,C 180.000} C_DIS
CIRC {X -316.968,Y -17.983,Z -20.000,A 0.015,B 0.000,C 180.000},{X -318.352,Y -20.658,Z -20.000,A 0.015,B 0.000,C 180.000} C_DIS
CIRC {X -318.263,Y -22.837,Z -20.000,A 0.015,B 0.000,C -180.000},{X -316.361,Y -23.901,Z -20.000,A 0.015,B -0.000,C 180.000} C_DIS
LIN {X -77.172,Y -23.901,Z -20.000,A 0.015,B 0.000,C 180.000} C_DIS
CIRC {X -75.259,Y -22.832,Z -20.000,A 0.015,B -0.000,C 180.000},{X -75.167,Y -20.643,Z -20.000,A 0.015,B 0.000,C 180.000} C_DIS
CIRC {X -76.785,Y -17.345,Z -20.000,A 0.015,B 0.000,C -180.000},{X -78.325,Y -14.010,Z -20.000,A 0.015,B 0.000,C 180.000} C_DIS
CIRC {X -79.569,Y -10.542,Z -20.000,A 0.015,B 0.000,C -180.000},{X -80.270,Y -6.925,Z -20.000,A 0.015,B -0.000,C -180.000} C_DIS
CIRC {X -79.431,Y 8.778,Z -20.000,A 0.015,B 0.000,C -180.000},{X -73.457,Y 23.325,Z -20.000,A 0.015,B 0.000,C 180.000} C_DIS
CIRC {X -65.362,Y 36.548,Z -20.000,A 0.015,B 0.000,C -180.000},{X -57.491,Y 49.907,Z -20.000,A 0.015,B 0.000,C -180.000} C_DIS
CIRC {X -53.342,Y 55.607,Z -20.000,A 0.015,B 0.000,C -180.000},{X -48.094,Y 60.317,Z -20.000,A 0.015,B 0.000,C -180.000} C_DIS
CIRC {X -42.203,Y 64.137,Z -20.000,A 0.015,B 0.000,C 180.000},{X -35.954,Y 67.338,Z -20.000,A 0.015,B 0.000,C 180.000} C_DIS
CIRC {X -32.046,Y 68.670,Z -20.000,A 0.015,B 0.000,C -180.000},{X -27.959,Y 69.248,Z -20.000,A 0.015,B 0.000,C 180.000} C_DIS
CIRC {X -23.850,Y 69.361,Z -20.000,A 0.015,B 0.000,C -180.000},{X -19.740,Y 69.317,Z -20.000,A 0.015,B 0.000,C 180.000} C_DIS
CIRC {X -15.550,Y 68.839,Z -20.000,A 0.015,B 0.000,C 180.000},{X -11.497,Y 67.672,Z -20.000,A 0.015,B 0.000,C 180.000} C_DIS
CIRC {X -7.636,Y 66.001,Z -20.000,A 0.015,B -0.000,C 180.000},{X -3.939,Y 63.993,Z -20.000,A 0.015,B -0.000,C 180.000} C_DIS
CIRC {X -2.959,Y 63.327,Z -20.000,A 0.015,B 0.000,C 180.000},{X -2.059,Y 62.556,Z -20.000,A 0.015,B 0.000,C -180.000} C_DIS
CIRC {X -1.186,Y 61.756,Z -20.000,A 0.015,B 0.000,C 180.000},{X -0.279,Y 60.996,Z -20.000,A 0.015,B 0.000,C 180.000} C_DIS
CIRC {X 1.796,Y 60.759,Z -20.000,A 0.015,B 0.000,C -180.000},{X 2.908,Y 62.526,Z -20.000,A 0.015,B 0.000,C 180.000} C_DIS
LIN {X 2.900,Y 327.991,Z -20.000,A 0.015,B 0.000,C 180.000} C_DIS
CIRC {X 1.772,Y 330.715,Z -20.000,A 0.015,B 0.000,C -180.000},{X -0.953,Y 331.844,Z -20.000,A 0.015,B 0.000,C -180.000} C_DIS
LIN {X -150.136,Y 331.840,Z -20.000,A 0.015,B 0.000,C 180.000} C_DIS
CIRC {X -151.781,Y 330.732,Z -20.000,A 0.015,B -0.000,C -180.000},{X -151.372,Y 328.790,Z -20.000,A 0.015,B 0.000,C 180.000} C_DIS
CIRC {X -148.252,Y 325.364,Z -20.000,A 0.015,B 0.000,C 180.000},{X -145.575,Y 321.582,Z -20.000,A 0.015,B -0.000,C -180.000} C_DIS
CIRC {X -143.365,Y 317.511,Z -20.000,A 0.015,B 0.000,C -180.000},{X -141.629,Y 313.216,Z -20.000,A 0.015,B 0.000,C -180.000} C_DIS
CIRC {X -140.498,Y 309.454,Z -20.000,A 0.015,B -0.000,C -180.000},{X -139.635,Y 305.622,Z -20.000,A 0.015,B -0.000,C 180.000} C_DIS
CIRC {X -139.136,Y 301.722,Z -20.000,A 0.015,B 0.000,C -180.000},{X -139.097,Y 297.790,Z -20.000,A 0.015,B 0.000,C 180.000} C_DIS
CIRC {X -142.600,Y 283.119,Z -20.000,A 0.015,B -0.000,C 180.000},{X -151.189,Y 270.719,Z -20.000,A 0.015,B -0.000,C 180.000} C_DIS
CIRC {X -163.792,Y 262.382,Z -20.000,A 0.015,B 0.000,C 180.000},{X -178.617,Y 259.457,Z -20.000,A 0.015,B -0.000,C -180.000} C_DIS
LIN {X -220.025,Y 260.044,Z -20.000,A 0.015,B 0.000,C 180.000} C_DIS
CIRC {X -228.536,Y 262.252,Z -20.000,A 0.015,B 0.000,C -180.000},{X -236.275,Y 266.424,Z -20.000,A 0.015,B 0.000,C 180.000} C_DIS
CIRC {X -242.975,Y 272.068,Z -20.000,A 0.015,B -0.000,C -180.000},{X -248.621,Y 278.767,Z -20.000,A 0.015,B -0.000,C -180.000} C_DIS
CIRC {X -250.810,Y 282.620,Z -20.000,A 0.015,B 0.000,C 180.000},{X -252.203,Y 286.828,Z -20.000,A 0.015,B 0.000,C -180.000} C_DIS
LIN {X -254.154,Y 295.499,Z -20.000,A 0.015,B -0.000,C -180.000} C_DIS
CIRC {X -254.564,Y 299.209,Z -20.000,A 0.015,B 0.000,C 180.000},{X -254.146,Y 302.917,Z -20.000,A 0.015,B 0.000,C 180.000} C_DIS
CIRC {X -253.389,Y 306.549,Z -20.000,A 0.015,B -0.000,C -180.000},{X -252.763,Y 310.205,Z -20.000,A 0.015,B 0.000,C -180.000} C_DIS
CIRC {X -251.513,Y 314.782,Z -20.000,A 0.015,B -0.000,C 180.000},{X -249.256,Y 318.954,Z -20.000,A 0.015,B 0.000,C -180.000} C_DIS
CIRC {X -248.819,Y 319.581,Z -20.000,A 0.015,B 0.000,C -180.000},{X -248.384,Y 320.208,Z -20.000,A 0.015,B 0.000,C 180.000} C_DIS
LIN {X -248.229,Y 320.817,Z -19.830,A 0.015,B 0.000,C 180.000} C_DIS
LIN {X -248.313,Y 321.272,Z -19.365,A 0.015,B 0.000,C -180.000} C_DIS
LIN {X -248.384,Y 321.426,Z -18.730,A 0.015,B 0.000,C -180.000} C_DIS
$VEL.CP = 1.00000
LIN {X -248.384,Y 321.426,Z 11.000,A 0.015,B -0.000,C 180.000} C_DIS
$VEL.CP = 1.00000
LIN {X -398.501,Y 339.199,Z 11.000,A 0.015,B -0.000,C 180.000} C_DIS
$VEL.CP = 1.00000
LIN {X -398.501,Y 339.199,Z 1.769,A 0.015,B -0.000,C -180.000} C_DIS
$VEL.CP = 0.10000
LIN {X -398.507,Y 339.199,Z 1.655,A 0.015,B -0.000,C -180.000} C_DIS
LIN {X -398.638,Y 339.197,Z 1.196,A 0.015,B 0.000,C -180.000} C_DIS
LIN {X -398.929,Y 339.182,Z 0.819,A 0.015,B -0.000,C -180.000} C_DIS
LIN {X -399.336,Y 339.133,Z 0.575,A 0.015,B 0.000,C -180.000} C_DIS
LIN {X -399.692,Y 339.076,Z 0.501,A 0.015,B -0.000,C 180.000} C_DIS
LIN {X -399.719,Y 339.072,Z 0.500,A 0.015,B 0.000,C 180.000} C_DIS
LIN {X -400.552,Y 338.848,Z 0.470,A 0.015,B 0.000,C 180.000} C_DIS
LIN {X -400.596,Y 338.832,Z 0.468,A 0.015,B -0.000,C -180.000} C_DIS
LIN {X -401.281,Y 338.494,Z 0.441,A 0.015,B -0.000,C -180.000} C_DIS
LIN {X -401.404,Y 338.418,Z 0.436,A 0.015,B 0.000,C 180.000} C_DIS
LIN {X -402.842,Y 337.053,Z 0.367,A 0.015,B -0.000,C -180.000} C_DIS
LIN {X -402.866,Y 337.018,Z 0.365,A 0.015,B -0.000,C -180.000} C_DIS
LIN {X -403.753,Y 334.430,Z 0.268,A 0.015,B 0.000,C -180.000} C_DIS
LIN {X -403.779,Y 333.946,Z 0.252,A 0.015,B 0.000,C 180.000} C_DIS
LIN {X -403.787,Y 333.653,Z 0.241,A 0.015,B 0.000,C 180.000} C_DIS
LIN {X -403.787,Y 333.050,Z 0.220,A 0.015,B 0.000,C 180.000} C_DIS
LIN {X -401.252,Y 328.076,Z 0.018,A 0.015,B -0.000,C -180.000} C_DIS
LIN {X -395.738,Y 327.203,Z -0.185,A 0.015,B 0.000,C 180.000} C_DIS
LIN {X -391.790,Y 331.150,Z -0.387,A 0.015,B -0.000,C -180.000} C_DIS
LIN {X -392.664,Y 336.664,Z -0.589,A 0.015,B 0.000,C -180.000} C_DIS
LIN {X -397.638,Y 339.199,Z -0.792,A 0.015,B 0.000,C 180.000} C_DIS
LIN {X -398.507,Y 339.199,Z -0.822,A 0.015,B 0.000,C 180.000} C_DIS
LIN {X -399.336,Y 339.133,Z -0.851,A 0.015,B 0.000,C -180.000} C_DIS
LIN {X -399.692,Y 339.076,Z -0.864,A 0.015,B 0.000,C 180.000} C_DIS
LIN {X -400.552,Y 338.848,Z -0.895,A 0.015,B -0.000,C -180.000} C_DIS
LIN {X -400.596,Y 338.832,Z -0.896,A 0.015,B 0.000,C -180.000} C_DIS
LIN {X -401.281,Y 338.494,Z -0.923,A 0.015,B 0.000,C 180.000} C_DIS
LIN {X -401.404,Y 338.418,Z -0.928,A 0.015,B 0.000,C -180.000} C_DIS
LIN {X -402.842,Y 337.053,Z -0.998,A 0.015,B -0.000,C -180.000} C_DIS
LIN {X -402.866,Y 337.018,Z -0.999,A 0.015,B 0.000,C -180.000} C_DIS
LIN {X -403.753,Y 334.430,Z -1.096,A 0.015,B 0.000,C -180.000} C_DIS
LIN {X -403.779,Y 333.946,Z -1.113,A 0.015,B -0.000,C -180.000} C_DIS
LIN {X -403.787,Y 333.653,Z -1.123,A 0.015,B 0.000,C -180.000} C_DIS
LIN {X -403.787,Y 333.050,Z -1.144,A 0.015,B 0.000,C 180.000} C_DIS
LIN {X -401.252,Y 328.076,Z -1.347,A 0.015,B 0.000,C -180.000} C_DIS
LIN {X -395.738,Y 327.203,Z -1.549,A 0.015,B -0.000,C -180.000} C_DIS
LIN {X -391.790,Y 331.150,Z -1.751,A 0.015,B 0.000,C -180.000} C_DIS
LIN {X -392.664,Y 336.664,Z -1.954,A 0.015,B 0.000,C -180.000} C_DIS
LIN {X -397.638,Y 339.199,Z -2.156,A 0.015,B 0.000,C -180.000} C_DIS
LIN {X -398.507,Y 339.199,Z -2.186,A 0.015,B -0.000,C -180.000} C_DIS
LIN {X -399.336,Y 339.133,Z -2.216,A 0.015,B -0.000,C 180.000} C_DIS
LIN {X -399.692,Y 339.076,Z -2.228,A 0.015,B 0.000,C -180.000} C_DIS
LIN {X -400.552,Y 338.848,Z -2.259,A 0.015,B 0.000,C -180.000} C_DIS
LIN {X -400.596,Y 338.832,Z -2.261,A 0.015,B 0.000,C -180.000} C_DIS
LIN {X -401.281,Y 338.494,Z -2.288,A 0.015,B -0.000,C -180.000} C_DIS
LIN {X -401.404,Y 338.418,Z -2.293,A 0.015,B 0.000,C -180.000} C_DIS
LIN {X -402.842,Y 337.053,Z -2.362,A 0.015,B 0.000,C -180.000} C_DIS
LIN {X -402.866,Y 337.018,Z -2.364,A 0.015,B 0.000,C -180.000} C_DIS
LIN {X -403.753,Y 334.430,Z -2.461,A 0.015,B -0.000,C -180.000} C_DIS
LIN {X -403.779,Y 333.946,Z -2.478,A 0.015,B 0.000,C 180.000} C_DIS
LIN {X -403.787,Y 333.653,Z -2.488,A 0.015,B -0.000,C -180.000} C_DIS
LIN {X -403.787,Y 333.050,Z -2.509,A 0.015,B -0.000,C -180.000} C_DIS
LIN {X -401.252,Y 328.076,Z -2.711,A 0.015,B 0.000,C -180.000} C_DIS
LIN {X -395.738,Y 327.203,Z -2.914,A 0.015,B 0.000,C -180.000} C_DIS
LIN {X -391.790,Y 331.150,Z -3.116,A 0.015,B 0.000,C 180.000} C_DIS
LIN {X -392.664,Y 336.664,Z -3.318,A 0.015,B -0.000,C -180.000} C_DIS
LIN {X -397.638,Y 339.199,Z -3.521,A 0.015,B -0.000,C -180.000} C_DIS
LIN {X -398.507,Y 339.199,Z -3.551,A 0.015,B -0.000,C -180.000} C_DIS
LIN {X -399.336,Y 339.133,Z -3.580,A 0.015,B 0.000,C -180.000} C_DIS
LIN {X -399.692,Y 339.076,Z -3.593,A 0.015,B -0.000,C -180.000} C_DIS
LIN {X -400.552,Y 338.848,Z -3.624,A 0.015,B -0.000,C -180.000} C_DIS
LIN {X -400.596,Y 338.832,Z -3.625,A 0.015,B -0.000,C -180.000} C_DIS
LIN {X -401.281,Y 338.494,Z -3.652,A 0.015,B 0.000,C -180.000} C_DIS
LIN {X -401.404,Y 338.418,Z -3.657,A 0.015,B 0.000,C 180.000} C_DIS
LIN {X -402.842,Y 337.053,Z -3.727,A 0.015,B 0.000,C 180.000} C_DIS
LIN {X -402.866,Y 337.018,Z -3.728,A 0.015,B -0.000,C -180.000} C_DIS
LIN {X -403.753,Y 334.430,Z -3.825,A 0.015,B -0.000,C 180.000} C_DIS
LIN {X -403.779,Y 333.946,Z -3.842,A 0.015,B 0.000,C 180.000} C_DIS
LIN {X -403.787,Y 333.653,Z -3.852,A 0.015,B -0.000,C -180.000} C_DIS
LIN {X -403.787,Y 333.050,Z -3.873,A 0.015,B 0.000,C -180.000} C_DIS
LIN {X -401.252,Y 328.076,Z -4.076,A 0.015,B 0.000,C 180.000} C_DIS
LIN {X -395.738,Y 327.203,Z -4.278,A 0.015,B 0.000,C 180.000} C_DIS
LIN {X -391.790,Y 331.150,Z -4.481,A 0.015,B 0.000,C 180.000} C_DIS
LIN {X -392.664,Y 336.664,Z -4.683,A 0.015,B -0.000,C -180.000} C_DIS
LIN {X -397.638,Y 339.199,Z -4.885,A 0.015,B 0.000,C -180.000} C_DIS
LIN {X -398.507,Y 339.199,Z -4.916,A 0.015,B 0.000,C 180.000} C_DIS
LIN {X -399.336,Y 339.133,Z -4.945,A 0.015,B 0.000,C -180.000} C_DIS
LIN {X -399.692,Y 339.076,Z -4.957,A 0.015,B 0.000,C -180.000} C_DIS
LIN {X -400.552,Y 338.848,Z -4.988,A 0.015,B 0.000,C 180.000} C_DIS
LIN {X -400.596,Y 338.832,Z -4.990,A 0.015,B 0.000,C -180.000} C_DIS
LIN {X -401.281,Y 338.494,Z -5.017,A 0.015,B -0.000,C -180.000} C_DIS
LIN {X -401.404,Y 338.418,Z -5.022,A 0.015,B -0.000,C 180.000} C_DIS
LIN {X -402.842,Y 337.053,Z -5.091,A 0.015,B 0.000,C 180.000} C_DIS
LIN {X -402.866,Y 337.018,Z -5.093,A 0.015,B 0.000,C 180.000} C_DIS
LIN {X -403.753,Y 334.430,Z -5.190,A 0.015,B 0.000,C -180.000} C_DIS
LIN {X -403.779,Y 333.946,Z -5.207,A 0.015,B -0.000,C -180.000} C_DIS
LIN {X -403.787,Y 333.653,Z -5.217,A 0.015,B -0.000,C -180.000} C_DIS
LIN {X -403.787,Y 333.050,Z -5.238,A 0.015,B -0.000,C -180.000} C_DIS
LIN {X -401.252,Y 328.076,Z -5.440,A 0.015,B 0.000,C -180.000} C_DIS
LIN {X -395.738,Y 327.203,Z -5.643,A 0.015,B -0.000,C -180.000} C_DIS
LIN {X -391.790,Y 331.150,Z -5.845,A 0.015,B 0.000,C -180.000} C_DIS
LIN {X -392.664,Y 336.664,Z -6.047,A 0.015,B 0.000,C -180.000} C_DIS
LIN {X -397.638,Y 339.199,Z -6.250,A 0.015,B 0.000,C -180.000} C_DIS
LIN {X -398.507,Y 339.199,Z -6.280,A 0.015,B 0.000,C 180.000} C_DIS
LIN {X -399.336,Y 339.133,Z -6.309,A 0.015,B -0.000,C 180.000} C_DIS
LIN {X -399.692,Y 339.076,Z -6.322,A 0.015,B 0.000,C -180.000} C_DIS
LIN {X -400.552,Y 338.848,Z -6.353,A 0.015,B 0.000,C 180.000} C_DIS
LIN {X -400.596,Y 338.832,Z -6.355,A 0.015,B -0.000,C 180.000} C_DIS
LIN {X -401.281,Y 338.494,Z -6.381,A 0.015,B -0.000,C -180.000} C_DIS
LIN {X -401.404,Y 338.418,Z -6.386,A 0.015,B -0.000,C 180.000} C_DIS
LIN {X -402.842,Y 337.053,Z -6.456,A 0.015,B -0.000,C -180.000} C_DIS
LIN {X -402.866,Y 337.018,Z -6.458,A 0.015,B 0.000,C -180.000} C_DIS
LIN {X -403.753,Y 334.430,Z -6.554,A 0.015,B 0.000,C 180.000} C_DIS
LIN {X -403.779,Y 333.946,Z -6.571,A 0.015,B -0.000,C -180.000} C_DIS
LIN {X -403.787,Y 333.653,Z -6.581,A 0.015,B -0.000,C 180.000} C_DIS
LIN {X -403.787,Y 333.050,Z -6.603,A 0.015,B 0.000,C -180.000} C_DIS
LIN {X -401.252,Y 328.076,Z -6.805,A 0.015,B -0.000,C -180.000} C_DIS
LIN {X -395.738,Y 327.203,Z -7.007,A 0.015,B 0.000,C 180.000} C_DIS
LIN {X -391.790,Y 331.150,Z -7.210,A 0.015,B 0.000,C -180.000} C_DIS
LIN {X -392.664,Y 336.664,Z -7.412,A 0.015,B -0.000,C -180.000} C_DIS
LIN {X -397.638,Y 339.199,Z -7.614,A 0.015,B 0.000,C -180.000} C_DIS
LIN {X -398.507,Y 339.199,Z -7.645,A 0.015,B 0.000,C 180.000} C_DIS
LIN {X -399.336,Y 339.133,Z -7.674,A 0.015,B 0.000,C -180.000} C_DIS
LIN {X -399.692,Y 339.076,Z -7.686,A 0.015,B -0.000,C -180.000} C_DIS
LIN {X -400.552,Y 338.848,Z -7.717,A 0.015,B -0.000,C 180.000} C_DIS
LIN {X -400.596,Y 338.832,Z -7.719,A 0.015,B -0.000,C -180.000} C_DIS
LIN {X -401.281,Y 338.494,Z -7.746,A 0.015,B -0.000,C -180.000} C_DIS
LIN {X -401.404,Y 338.418,Z -7.751,A 0.015,B -0.000,C -180.000} C_DIS
LIN {X -402.842,Y 337.053,Z -7.821,A 0.015,B 0.000,C -180.000} C_DIS
LIN {X -402.866,Y 337.018,Z -7.822,A 0.015,B -0.000,C -180.000} C_DIS
LIN {X -403.753,Y 334.430,Z -7.919,A 0.015,B -0.000,C -180.000} C_DIS
LIN {X -403.779,Y 333.946,Z -7.936,A 0.015,B 0.000,C 180.000} C_DIS
LIN {X -403.787,Y 333.653,Z -7.946,A 0.015,B 0.000,C -180.000} C_DIS
LIN {X -403.787,Y 333.050,Z -7.967,A 0.015,B 0.000,C 180.000} C_DIS
LIN {X -401.252,Y 328.076,Z -8.169,A 0.015,B 0.000,C -180.000} C_DIS
LIN {X -395.738,Y 327.203,Z -8.372,A 0.015,B 0.000,C 180.000} C_DIS
LIN {X -391.790,Y 331.150,Z -8.574,A 0.015,B -0.000,C -180.000} C_DIS
LIN {X -392.664,Y 336.664,Z -8.777,A 0.015,B -0.000,C -180.000} C_DIS
LIN {X -397.638,Y 339.199,Z -8.979,A 0.015,B -0.000,C -180.000} C_DIS
LIN {X -398.507,Y 339.199,Z -9.009,A 0.015,B 0.000,C -180.000} C_DIS
LIN {X -399.336,Y 339.133,Z -9.038,A 0.015,B 0.000,C -180.000} C_DIS
LIN {X -399.692,Y 339.076,Z -9.051,A 0.015,B 0.000,C 180.000} C_DIS
LIN {X -400.552,Y 338.848,Z -9.082,A 0.015,B 0.000,C -180.000} C_DIS
LIN {X -400.596,Y 338.832,Z -9.084,A 0.015,B 0.000,C 180.000} C_DIS
LIN {X -401.281,Y 338.494,Z -9.110,A 0.015,B -0.000,C -180.000} C_DIS
LIN {X -401.404,Y 338.418,Z -9.115,A 0.015,B 0.000,C -180.000} C_DIS
LIN {X -402.842,Y 337.053,Z -9.185,A 0.015,B 0.000,C -180.000} C_DIS
LIN {X -402.866,Y 337.018,Z -9.187,A 0.015,B -0.000,C -180.000} C_DIS
LIN {X -403.753,Y 334.430,Z -9.283,A 0.015,B 0.000,C 180.000} C_DIS
LIN {X -403.779,Y 333.946,Z -9.300,A 0.015,B 0.000,C -180.000} C_DIS
LIN {X -403.787,Y 333.653,Z -9.311,A 0.015,B 0.000,C -180.000} C_DIS
LIN {X -403.787,Y 333.050,Z -9.332,A 0.015,B 0.000,C 180.000} C_DIS
LIN {X -401.252,Y 328.076,Z -9.534,A 0.015,B -0.000,C 180.000} C_DIS
LIN {X -395.738,Y 327.203,Z -9.736,A 0.015,B 0.000,C -180.000} C_DIS
LIN {X -391.790,Y 331.150,Z -9.939,A 0.015,B 0.000,C 180.000} C_DIS
LIN {X -392.664,Y 336.664,Z -10.141,A 0.015,B -0.000,C 180.000} C_DIS
LIN {X -397.638,Y 339.199,Z -10.343,A 0.015,B -0.000,C -180.000} C_DIS
LIN {X -398.507,Y 339.199,Z -10.374,A 0.015,B -0.000,C -180.000} C_DIS
LIN {X -399.336,Y 339.133,Z -10.403,A 0.015,B -0.000,C -180.000} C_DIS
LIN {X -399.692,Y 339.076,Z -10.415,A 0.015,B 0.000,C 180.000} C_DIS
LIN {X -400.552,Y 338.848,Z -10.447,A 0.015,B -0.000,C -180.000} C_DIS
LIN {X -400.596,Y 338.832,Z -10.448,A 0.015,B -0.000,C 180.000} C_DIS
LIN {X -401.281,Y 338.494,Z -10.475,A 0.015,B -0.000,C -180.000} C_DIS
LIN {X -401.404,Y 338.418,Z -10.480,A 0.015,B -0.000,C -180.000} C_DIS
LIN {X -402.842,Y 337.053,Z -10.550,A 0.015,B -0.000,C -180.000} C_DIS
LIN {X -402.866,Y 337.018,Z -10.551,A 0.015,B 0.000,C 180.000} C_DIS
LIN {X -403.753,Y 334.430,Z -10.648,A 0.015,B 0.000,C -180.000} C_DIS
LIN {X -403.779,Y 333.946,Z -10.665,A 0.015,B -0.000,C -180.000} C_DIS
LIN {X -403.787,Y 333.653,Z -10.675,A 0.015,B -0.000,C -180.000} C_DIS
LIN {X -403.787,Y 333.050,Z -10.696,A 0.015,B -0.000,C -180.000} C_DIS
LIN {X -401.252,Y 328.076,Z -10.899,A 0.015,B 0.000,C -180.000} C_DIS
LIN {X -395.738,Y 327.203,Z -11.101,A 0.015,B 0.000,C -180.000} C_DIS
LIN {X -391.790,Y 331.150,Z -11.303,A 0.015,B -0.000,C -180.000} C_DIS
LIN {X -392.664,Y 336.664,Z -11.506,A 0.015,B 0.000,C -180.000} C_DIS
LIN {X -397.638,Y 339.199,Z -11.708,A 0.015,B -0.000,C 180.000} C_DIS
LIN {X -398.507,Y 339.199,Z -11.738,A 0.015,B -0.000,C 180.000} C_DIS
LIN {X -399.336,Y 339.133,Z -11.767,A 0.015,B -0.000,C 180.000} C_DIS
LIN {X -399.692,Y 339.076,Z -11.780,A 0.015,B 0.000,C -180.000} C_DIS
LIN {X -400.552,Y 338.848,Z -11.811,A 0.015,B -0.000,C -180.000} C_DIS
LIN {X -400.596,Y 338.832,Z -11.813,A 0.015,B 0.000,C 180.000} C_DIS
LIN {X -401.281,Y 338.494,Z -11.839,A 0.015,B 0.000,C 180.000} C_DIS
LIN {X -401.404,Y 338.418,Z -11.844,A 0.015,B -0.000,C -180.000} C_DIS
LIN {X -402.842,Y 337.053,Z -11.914,A 0.015,B -0.000,C -180.000} C_DIS
LIN {X -402.866,Y 337.018,Z -11.916,A 0.015,B -0.000,C -180.000} C_DIS
LIN {X -403.753,Y 334.430,Z -12.012,A 0.015,B 0.000,C -180.000} C_DIS
LIN {X -403.779,Y 333.946,Z -12.029,A 0.015,B -0.000,C 180.000} C_DIS
LIN {X -403.787,Y 333.653,Z -12.040,A 0.015,B -0.000,C -180.000} C_DIS
LIN {X -403.787,Y 333.050,Z -12.061,A 0.015,B 0.000,C 180.000} C_DIS
LIN {X -401.252,Y 328.076,Z -12.263,A 0.015,B -0.000,C -180.000} C_DIS
LIN {X -395.738,Y 327.203,Z -12.465,A 0.015,B 0.000,C -180.000} C_DIS
LIN {X -391.790,Y 331.150,Z -12.668,A 0.015,B -0.000,C -180.000} C_DIS
LIN {X -392.664,Y 336.664,Z -12.870,A 0.015,B 0.000,C 180.000} C_DIS
LIN {X -397.638,Y 339.199,Z -13.073,A 0.015,B 0.000,C -180.000} C_DIS
LIN {X -398.507,Y 339.199,Z -13.103,A 0.015,B -0.000,C 180.000} C_DIS
LIN {X -399.336,Y 339.133,Z -13.132,A 0.015,B -0.000,C -180.000} C_DIS
LIN {X -399.692,Y 339.076,Z -13.145,A 0.015,B 0.000,C -180.000} C_DIS
LIN {X -400.552,Y 338.848,Z -13.176,A 0.015,B 0.000,C -180.000} C_DIS
LIN {X -400.596,Y 338.832,Z -13.177,A 0.015,B -0.000,C -180.000} C_DIS
LIN {X -401.281,Y 338.494,Z -13.204,A 0.015,B 0.000,C -180.000} C_DIS
LIN {X -401.404,Y 338.418,Z -13.209,A 0.015,B 0.000,C -180.000} C_DIS
LIN {X -402.842,Y 337.053,Z -13.279,A 0.015,B 0.000,C -180.000} C_DIS
LIN {X -402.866,Y 337.018,Z -13.280,A 0.015,B 0.000,C 180.000} C_DIS
LIN {X -403.753,Y 334.430,Z -13.377,A 0.015,B 0.000,C 180.000} C_DIS
LIN {X -403.779,Y 333.946,Z -13.394,A 0.015,B 0.000,C -180.000} C_DIS
LIN {X -403.787,Y 333.653,Z -13.404,A 0.015,B -0.000,C 180.000} C_DIS
LIN {X -403.787,Y 333.050,Z -13.425,A 0.015,B 0.000,C 180.000} C_DIS
LIN {X -401.252,Y 328.076,Z -13.628,A 0.015,B 0.000,C -180.000} C_DIS
LIN {X -395.738,Y 327.203,Z -13.830,A 0.015,B 0.000,C -180.000} C_DIS
LIN {X -391.790,Y 331.150,Z -14.032,A 0.015,B -0.000,C -180.000} C_DIS
LIN {X -392.664,Y 336.664,Z -14.235,A 0.015,B -0.000,C 180.000} C_DIS
LIN {X -397.638,Y 339.199,Z -14.437,A 0.015,B 0.000,C -180.000} C_DIS
LIN {X -398.507,Y 339.199,Z -14.467,A 0.015,B 0.000,C -180.000} C_DIS
LIN {X -399.336,Y 339.133,Z -14.496,A 0.015,B 0.000,C 180.000} C_DIS
LIN {X -399.692,Y 339.076,Z -14.509,A 0.015,B -0.000,C 180.000} C_DIS
LIN {X -400.552,Y 338.848,Z -14.540,A 0.015,B -0.000,C -180.000} C_DIS
LIN {X -400.596,Y 338.832,Z -14.542,A 0.015,B -0.000,C 180.000} C_DIS
LIN {X -401.281,Y 338.494,Z -14.569,A 0.015,B 0.000,C -180.000} C_DIS
LIN {X -401.404,Y 338.418,Z -14.574,A 0.015,B -0.000,C -180.000} C_DIS
LIN {X -402.842,Y 337.053,Z -14.643,A 0.015,B 0.000,C -180.000} C_DIS
LIN {X -402.866,Y 337.018,Z -14.645,A 0.015,B 0.000,C 180.000} C_DIS
LIN {X -403.753,Y 334.430,Z -14.742,A 0.015,B -0.000,C -180.000} C_DIS
LIN {X -403.779,Y 333.946,Z -14.758,A 0.015,B 0.000,C -180.000} C_DIS
LIN {X -403.787,Y 333.653,Z -14.769,A 0.015,B 0.000,C -180.000} C_DIS
LIN {X -403.787,Y 333.050,Z -14.790,A 0.015,B 0.000,C -180.000} C_DIS
LIN {X -401.252,Y 328.076,Z -14.992,A 0.015,B -0.000,C -180.000} C_DIS
LIN {X -395.738,Y 327.203,Z -15.195,A 0.015,B 0.000,C 180.000} C_DIS
LIN {X -391.790,Y 331.150,Z -15.397,A 0.015,B 0.000,C 180.000} C_DIS
LIN {X -392.664,Y 336.664,Z -15.599,A 0.015,B -0.000,C -180.000} C_DIS
LIN {X -397.638,Y 339.199,Z -15.802,A 0.015,B -0.000,C -180.000} C_DIS
LIN {X -398.507,Y 339.199,Z -15.832,A 0.015,B 0.000,C 180.000} C_DIS
LIN {X -399.336,Y 339.133,Z -15.861,A 0.015,B 0.000,C -180.000} C_DIS
LIN {X -399.692,Y 339.076,Z -15.874,A 0.015,B 0.000,C -180.000} C_DIS
LIN {X -400.552,Y 338.848,Z -15.905,A 0.015,B -0.000,C -180.000} C_DIS
LIN {X -400.596,Y 338.832,Z -15.906,A 0.015,B -0.000,C 180.000} C_DIS
LIN {X -401.281,Y 338.494,Z -15.933,A 0.015,B 0.000,C 180.000} C_DIS
LIN {X -401.404,Y 338.418,Z -15.938,A 0.015,B 0.000,C -180.000} C_DIS
LIN {X -402.842,Y 337.053,Z -16.008,A 0.015,B 0.000,C -180.000} C_DIS
LIN {X -402.866,Y 337.018,Z -16.009,A 0.015,B 0.000,C -180.000} C_DIS
LIN {X -403.753,Y 334.430,Z -16.106,A 0.015,B -0.000,C -180.000} C_DIS
LIN {X -403.779,Y 333.946,Z -16.123,A 0.015,B -0.000,C 180.000} C_DIS
LIN {X -403.787,Y 333.653,Z -16.133,A 0.015,B -0.000,C -180.000} C_DIS
LIN {X -403.787,Y 333.050,Z -16.154,A 0.015,B 0.000,C 180.000} C_DIS
LIN {X -401.252,Y 328.076,Z -16.357,A 0.015,B -0.000,C 180.000} C_DIS
LIN {X -395.738,Y 327.203,Z -16.559,A 0.015,B 0.000,C -180.000} C_DIS
LIN {X -391.790,Y 331.150,Z -16.761,A 0.015,B 0.000,C -180.000} C_DIS
LIN {X -392.664,Y 336.664,Z -16.964,A 0.015,B -0.000,C -180.000} C_DIS
LIN {X -397.638,Y 339.199,Z -17.166,A 0.015,B -0.000,C -180.000} C_DIS
LIN {X -398.507,Y 339.199,Z -17.196,A 0.015,B -0.000,C 180.000} C_DIS
LIN {X -399.336,Y 339.133,Z -17.226,A 0.015,B 0.000,C 180.000} C_DIS
LIN {X -399.692,Y 339.076,Z -17.238,A 0.015,B -0.000,C 180.000} C_DIS
LIN {X -400.552,Y 338.848,Z -17.269,A 0.015,B 0.000,C 180.000} C_DIS
LIN {X -400.596,Y 338.832,Z -17.271,A 0.015,B 0.000,C -180.000} C_DIS
LIN {X -401.281,Y 338.494,Z -17.298,A 0.015,B -0.000,C -180.000} C_DIS
LIN {X -401.404,Y 338.418,Z -17.303,A 0.015,B -0.000,C -180.000} C_DIS
LIN {X -402.842,Y 337.053,Z -17.372,A 0.015,B -0.000,C -180.000} C_DIS
LIN {X -402.866,Y 337.018,Z -17.374,A 0.015,B -0.000,C -180.000} C_DIS
LIN {X -403.753,Y 334.430,Z -17.471,A 0.015,B -0.000,C -180.000} C_DIS
LIN {X -403.779,Y 333.946,Z -17.488,A 0.015,B 0.000,C 180.000} C_DIS
LIN {X -403.787,Y 333.653,Z -17.498,A 0.015,B -0.000,C -180.000} C_DIS
